(* CODESYS project PLC.project

Project tree, tasks and I/O mapping:
  A_SIM : CODESYS Control Win V3, 3S - Smart Software Solutions GmbH, order no. 305021, version 3.5.10.70
    application PE
      libraries: Standard, * (System); MemoryUtils, * (3S - Smart Software Solutions GmbH); SysTime, 3.5.9.0 (System); PE Core, 0.0.0.23 (ProdexSys); PE User, 0.0.0.15 (ProdexSys)
      task DB (cyclic, interval t#10ms, priority 1) calls DB
      task C100MS (cyclic, interval t#100ms, priority 2) calls C100MS
      task FreeWheel (freewheeling, priority 31) calls SYS, MAIN
      Symbols
      global variables GC
      global variables GVL
      program C100MS [ST]
      program DB [ST]
      program MAIN [ST]: hcb, states, hrb
      program SYS [ST]: updatePointers, initTypes, updateHW, exReadTagsCall, exWriteTagsCall, templateMonitor
      GlobalTypes/
        data type HW
        data type Instances
        data type M
        data type TemplateInstances
        data type TemplateInstancesM
        data type Instructions
        EX/
          data type Exchange
          States/
            data type ValveRegStates
            data type GasFlowRegStates
            data type DriveStates
            data type DriveRegStates
            data type DigOutStates
            data type SensorDigStates
            data type SensorAnStates
            data type PidCStates
            data type HysteresisStates
            data type CascadeStates
            data type HysteresisExStates
            data type WindowExchange
            data type ValveStates
          HCB/
            data type HmiCmd
            data type HmiCmdBuffer
            data type ControlLoop
          HRB/
            data type HmiReadReq
            data type HmiReadRes
            data type HmiReadBuffer
        data type Descriptions
        data type TagsExM
  RLDA : RLDA ARM WinCE (NIL AP), RLDA, ltd., order no. 001, version 3.5.15.10
    application PE
      libraries: Standard, * (System); MemoryUtils, * (3S - Smart Software Solutions GmbH); SysTime, 3.5.9.0 (System); PE Core, 0.0.0.23 (ProdexSys); PE User, 0.0.0.15 (ProdexSys)
      task DB (cyclic, interval t#10ms, priority 1) calls DB
      task FreeWheel (freewheeling, priority 31) calls SYS, MAIN
      task C100MS (cyclic, interval t#100ms, priority 2) calls C100MS
      global variables GC
      global variables GVL
      program C100MS [ST]
      program DB [ST]
      program MAIN [ST]: hcb, states, hrb
      GlobalTypes/
        data type HW
        data type Instances
        data type M
        data type TemplateInstances
        data type TemplateInstancesM
        data type Instructions
        data type Descriptions
        data type TagsExM
        EX/
          data type Exchange
          HCB/
            data type HmiCmd
            data type HmiCmdBuffer
            data type ControlLoop
          HRB/
            data type HmiReadReq
            data type HmiReadRes
            data type HmiReadBuffer
          States/
            data type DriveStates
            data type DriveRegStates
            data type DigOutStates
            data type SensorDigStates
            data type SensorAnStates
            data type PidCStates
            data type HysteresisStates
            data type CascadeStates
            data type HysteresisExStates
            data type WindowExchange
            data type ValveStates
            data type ValveRegStates
            data type GasFlowRegStates
      program SYS [ST]: updateHW, updatePointers, exReadTagsCall, exWriteTagsCall, templateMonitor, initTypes
      Symbols
    Modbus_COM : Modbus COM, 3S - Smart Software Solutions GmbH, version 3.4.0.0
        settings: DataBits = 8; StopBits = 1; ComPort = 2
      Modbus_Master_COM_Port : Modbus Master, COM Port, 3S - Smart Software Solutions GmbH, version 3.5.10.30
        NL_S_16DI : NL(S)-16DI, RLDA, ltd., version 3.5.11.0
            settings: SlaveAddress = 11; ResponseTimeout = 500; UseExtendedFunctionCodes = TRUE
            unmapped channels: Channel 0
        NL_S_8AI_16ch : NL(S)-8AI_16ch, RLDA, ltd., version 3.5.11.0
            settings: SlaveAddress = 10; ResponseTimeout = 500; UseExtendedFunctionCodes = TRUE
            unmapped channels: Channel 0, Channel 1, Channel 2, Channel 3, Channel 4, Channel 5, Channel 6, Channel 7, Channel 8, Channel 9, Channel 10, Channel 11, Channel 12, Channel 13, Channel 14, Channel 15
*)

// A_SIM/PE/GlobalTypes/EX/States/ValveRegStates
TYPE ValveRegStates :
STRUCT
	status : ARRAY[0..GC.VALVE_REG_MAX_IDX]OF DWORD;
	sp : ARRAY[0..GC.VALVE_REG_MAX_IDX]OF REAL;
END_STRUCT
END_TYPE

// A_SIM/PE/GlobalTypes/EX/States/GasFlowRegStates
TYPE GasFlowRegStates :
STRUCT
	status : ARRAY[0..GC.GAS_FLOW_REG_MAX_IDX]OF DWORD;
	sp : ARRAY[0..GC.GAS_FLOW_REG_MAX_IDX]OF REAL;
	pv : ARRAY[0..GC.GAS_FLOW_REG_MAX_IDX]OF REAL;
END_STRUCT
END_TYPE

// A_SIM/PE/GlobalTypes/EX/States/DriveStates
TYPE DriveStates :
STRUCT
	status : ARRAY[0..GC.DRIVE_MAX_IDX]OF DWORD;
END_STRUCT
END_TYPE

// A_SIM/PE/GlobalTypes/EX/States/DriveRegStates
TYPE DriveRegStates :
STRUCT
	status : ARRAY[0..GC.DRIVE_REG_MAX_IDX]OF DWORD;
	sp : ARRAY[0..GC.DRIVE_REG_MAX_IDX]OF REAL;
	pv : ARRAY[0..GC.DRIVE_REG_MAX_IDX]OF REAL;
END_STRUCT
END_TYPE

// A_SIM/PE/GlobalTypes/EX/States/DigOutStates
TYPE DigOutStates :
STRUCT
	status : ARRAY[0..GC.DIG_OUT_MAX_IDX]OF DWORD;
END_STRUCT
END_TYPE

// A_SIM/PE/GlobalTypes/EX/States/SensorDigStates
TYPE SensorDigStates :
STRUCT
	status : ARRAY[0..GC.SENSOR_DIG_MAX_IDX]OF DWORD;
END_STRUCT
END_TYPE

// A_SIM/PE/GlobalTypes/EX/States/SensorAnStates
TYPE SensorAnStates :
STRUCT
	status : ARRAY[0..GC.SENSOR_AN_MAX_IDX]OF DWORD;
	sp : ARRAY[0..GC.SENSOR_AN_MAX_IDX]OF REAL;
	pv : ARRAY[0..GC.SENSOR_AN_MAX_IDX]OF REAL;
END_STRUCT
END_TYPE

// A_SIM/PE/GlobalTypes/EX/States/PidCStates
TYPE PidCStates :
STRUCT
	status : ARRAY[0..GC.PID_C_MAX_IDX]OF DWORD;
	out : ARRAY[0..GC.PID_C_MAX_IDX]OF REAL;
END_STRUCT
END_TYPE

// A_SIM/PE/GlobalTypes/EX/States/HysteresisStates
TYPE HysteresisStates :
STRUCT
	status : ARRAY[0..GC.HYSTERESIS_MAX_IDX]OF DWORD;
	out1 : ARRAY[0..GC.HYSTERESIS_MAX_IDX]OF BOOL;
	out2 : ARRAY[0..GC.HYSTERESIS_MAX_IDX]OF BOOL;
END_STRUCT
END_TYPE

// A_SIM/PE/GlobalTypes/EX/States/CascadeStates
TYPE CascadeStates :
STRUCT
	status : ARRAY[0..GC.REF_MAX_IDX]OF DWORD;
END_STRUCT
END_TYPE

// A_SIM/PE/GlobalTypes/EX/States/HysteresisExStates
TYPE HysteresisExStates :
STRUCT
	status : ARRAY[0..GC.HYSTERESISEX_MAX_IDX]OF DWORD;
	outActuator : ARRAY[0..GC.HYSTERESISEX_MAX_IDX,0..4]OF BOOL;
	out : ARRAY[0..GC.HYSTERESISEX_MAX_IDX]OF BOOL;
END_STRUCT
END_TYPE

// A_SIM/PE/GlobalTypes/EX/States/WindowExchange
TYPE WindowExchange :
STRUCT
	locks : ARRAY[0..GC.WINDOW_MAX_IDX]OF UDINT;
	errors : ARRAY[0..GC.WINDOW_MAX_IDX]OF UDINT;
	status : ARRAY[0..GC.WINDOW_MAX_IDX]OF UDINT;
	workTime : ARRAY[0..GC.WINDOW_MAX_IDX]OF TIME;
END_STRUCT
END_TYPE

// A_SIM/PE/GlobalTypes/HW
TYPE HW :
STRUCT
	di16: ARRAY[0..GC.DI16_MAX_IDX] OF PEU.DI16Instance;
	do16: ARRAY[0..GC.DO16_MAX_IDX] OF PEU.DO16Instance;
	ai16: ARRAY[0..GC.AI16_MAX_IDX] OF PEU.AI16Instance;
	ao4: ARRAY[0..GC.AO4_MAX_IDX] OF PEU.AO4Instance;
END_STRUCT
END_TYPE

// A_SIM/PE/GlobalTypes/Instances
TYPE Instances :
STRUCT
	template: ARRAY[0..PEC.GC.TEMPLATE_MAX_IDX]OF TemplateInstances;
	window : ARRAY[0..PEC.GC.WINDOW_MAX_IDX] OF PEC.WindowInstance;
	parameters : ARRAY[0..PEC.GC.PARAMETERS_MAX_IDX] OF PEC.ParametersInstance;	
	
	valve: ARRAY[0..GC.VALVE_MAX_IDX] OF PEU.ValveInstance;
	valveReg: ARRAY[0..GC.VALVE_REG_MAX_IDX] OF PEU.ValveRegInstance;
	drive: ARRAY[0..GC.DRIVE_MAX_IDX] OF PEU.DriveInstance;
	driveReg: ARRAY[0..GC.DRIVE_REG_MAX_IDX] OF PEU.DriveRegInstance;
	sensorDig : ARRAY[0..GC.SENSOR_DIG_MAX_IDX]OF SensorDigInstance;
	sensorAn : ARRAY[0..GC.SENSOR_AN_MAX_IDX]OF SensorAnInstance;
	pidC : ARRAY[0..GC.PID_C_MAX_IDX]OF PidCInstance;
	hysteresis : ARRAY[0..GC.HYSTERESIS_MAX_IDX]OF HysteresisInstance;
	gasFlowReg : ARRAY[0..GC.GAS_FLOW_REG_MAX_IDX]OF GasFlowRegInstance;
	cascade : ARRAY[0..GC.REF_MAX_IDX]OF CascadeInstance;
	dose : ARRAY[0..GC.DOSE_MAX_IDX]OF DoseInstance;
	profile : ARRAY[0..GC.PROFILE_MAX_IDX]OF ProfileInstance;
	ramp : ARRAY[0..GC.RAMP_MAX_IDX]OF RampInstance;
	route : ARRAY[0..GC.ROUTE_MAX_IDX]OF RouteInstance;
	flip : ARRAY[0..GC.FLIP_MAX_IDX]OF FlipInstance;
	digOut : ARRAY[0..GC.DIG_OUT_MAX_IDX]OF DigOutInstance;
	hysteresisEx : ARRAY[0..GC.HYSTERESISEX_MAX_IDX]OF HysteresisExInstance;
END_STRUCT
END_TYPE

// A_SIM/PE/GlobalTypes/M
TYPE M :
STRUCT
	template : ARRAY[0..PEC.GC.TEMPLATE_MAX_IDX]OF TemplateInstancesM;
	window : ARRAY[0..PEC.GC.WINDOW_MAX_IDX] OF PEC.WindowM;
	parameters : ARRAY[0..PEC.GC.PARAMETERS_MAX_IDX] OF PEC.ParametersM;
	rcpCommon : ARRAY[0..GC.RCP_CALL_INST_MAX_IDX] OF PEC.RcpCommonM;
	rcpStage : ARRAY[0..GC.RCP_CALL_INST_MAX_IDX] OF PEC.RcpStageM;
	rcpStep : ARRAY[0..GC.RCP_CALL_INST_MAX_IDX] OF PEC.RcpStepM;
	di16: ARRAY[0..GC.DI16_MAX_IDX] OF PEU.DI16M;
	do16: ARRAY[0..GC.DO16_MAX_IDX] OF PEU.DO16M;
	ai16: ARRAY[0..GC.AI16_MAX_IDX] OF PEU.AI16M;
	ao4: ARRAY[0..GC.AO4_MAX_IDX] OF PEU.AO4M;
	
	valve: ARRAY[0..GC.VALVE_MAX_IDX] OF PEU.ValveM;
	valveReg: ARRAY[0..GC.VALVE_REG_MAX_IDX] OF PEU.ValveRegM;
	drive: ARRAY[0..GC.DRIVE_MAX_IDX] OF PEU.DriveM;
	driveReg: ARRAY[0..GC.DRIVE_REG_MAX_IDX] OF PEU.DriveRegM;
	sensorDig : ARRAY[0..GC.SENSOR_DIG_MAX_IDX]OF SensorDigM;
	sensorAn : ARRAY[0..GC.SENSOR_AN_MAX_IDX]OF SensorAnM;
	pidC : ARRAY[0..GC.PID_C_MAX_IDX]OF PidCM;
	hysteresis : ARRAY[0..GC.HYSTERESIS_MAX_IDX]OF HysteresisM;
	gasFlowReg : ARRAY[0..GC.GAS_FLOW_REG_MAX_IDX]OF GasFlowRegM;
	cascade : ARRAY[0..GC.REF_MAX_IDX]OF CascadeM;
	dose : ARRAY[0..GC.DOSE_MAX_IDX]OF DoseM;
	profile : ARRAY[0..GC.PROFILE_MAX_IDX]OF ProfileM;
	ramp : ARRAY[0..GC.RAMP_MAX_IDX]OF RampM;
	route : ARRAY[0..GC.ROUTE_MAX_IDX]OF RouteM;
	flip : ARRAY[0..GC.FLIP_MAX_IDX]OF FlipM;
	digOut : ARRAY[0..GC.DIG_OUT_MAX_IDX]OF DigOutM;
	hysteresisEx : ARRAY[0..GC.HYSTERESISEX_MAX_IDX]OF HysteresisExM;
	area: ARRAY[0..GC.AREA_MAX_IDX] OF AreaM;
	
END_STRUCT
END_TYPE

// A_SIM/PE/GlobalTypes/TemplateInstances
TYPE TemplateInstances :
STRUCT
	instance : ARRAY[0..PEC.GC.TEMPLATE_INST_MAX_IDX] OF PEC.TemplateInstance;
END_STRUCT
END_TYPE

// A_SIM/PE/GlobalTypes/TemplateInstancesM
TYPE TemplateInstancesM :
STRUCT
	instance : ARRAY[0..PEC.GC.TEMPLATE_INST_MAX_IDX] OF TemplateInstM;
END_STRUCT
END_TYPE

// A_SIM/PE/GlobalTypes/Instructions
TYPE Instructions :
STRUCT
	edge : ARRAY[0..GC.IEDGE_M_MAX_IDX]OF PEC.IEdgeInstance;
	trig : ARRAY[0..GC.ITRIG_M_MAX_IDX]OF PEC.ITrigInstance;
	timer : ARRAY[0..GC.ITIMER_MAX_IDX]OF PEC.ITimerInstance;
	counter : ARRAY[0..GC.ICOUNTER_MAX_IDX]OF PEC.ICounterInstance;
	pulse : ARRAY[0..GC.IPULSE_MAX_IDX]OF PEC.IPulseInstance;
	rcpCommon : ARRAY[0..GC.RCP_CALL_INST_MAX_IDX] OF PEC.RcpCommonInstance;
	rcpStage : ARRAY[0..GC.RCP_CALL_INST_MAX_IDX] OF PEC.RcpStageInstance;
	rcpStep : ARRAY[0..GC.RCP_CALL_INST_MAX_IDX] OF PEC.RcpStepInstance;
END_STRUCT
END_TYPE

// A_SIM/PE/GlobalTypes/EX/States/ValveStates
TYPE ValveStates :
STRUCT
	status: ARRAY[0..GC.VALVE_MAX_IDX] OF DWORD;
END_STRUCT
END_TYPE

// A_SIM/PE/GlobalTypes/EX/Exchange
TYPE Exchange :
STRUCT	
	hcb: ARRAY[0..GC.HCB_MAX_IDX] OF HmiCmdBuffer;
	hrb: ARRAY[0..GC.HRB_MAX_IDX] OF HmiReadBuffer;
	window : WindowExchange;
	valve : ValveStates;
	valveReg : ValveRegStates;
	gasFlowReg : GasFlowRegStates;
	drive : DriveStates;
	driveReg : DriveRegStates;
	sensorDig : SensorDigStates;
	sensorAn : SensorAnStates;
	pidC : PidCStates;
	hysteresis : HysteresisStates;
	cascade : CascadeStates;
	digOut : DigOutStates;
	hysteresisEx : HysteresisExStates;
END_STRUCT
END_TYPE

// RLDA/PE/GlobalTypes/EX/States/DriveStates
TYPE DriveStates :
STRUCT
	status : ARRAY[0..GC.DRIVE_MAX_IDX]OF DWORD;
END_STRUCT
END_TYPE

// RLDA/PE/GlobalTypes/EX/States/DriveRegStates
TYPE DriveRegStates :
STRUCT
	status : ARRAY[0..GC.DRIVE_REG_MAX_IDX]OF DWORD;
	sp : ARRAY[0..GC.DRIVE_REG_MAX_IDX]OF REAL;
	pv : ARRAY[0..GC.DRIVE_REG_MAX_IDX]OF REAL;
END_STRUCT
END_TYPE

// RLDA/PE/GlobalTypes/EX/States/DigOutStates
TYPE DigOutStates :
STRUCT
	status : ARRAY[0..GC.DIG_OUT_MAX_IDX]OF DWORD;
END_STRUCT
END_TYPE

// RLDA/PE/GlobalTypes/EX/States/SensorDigStates
TYPE SensorDigStates :
STRUCT
	status : ARRAY[0..GC.SENSOR_DIG_MAX_IDX]OF DWORD;
END_STRUCT
END_TYPE

// RLDA/PE/GlobalTypes/EX/States/SensorAnStates
TYPE SensorAnStates :
STRUCT
	status : ARRAY[0..GC.SENSOR_AN_MAX_IDX]OF DWORD;
	sp : ARRAY[0..GC.SENSOR_AN_MAX_IDX]OF REAL;
	pv : ARRAY[0..GC.SENSOR_AN_MAX_IDX]OF REAL;
END_STRUCT
END_TYPE

// RLDA/PE/GlobalTypes/EX/States/PidCStates
TYPE PidCStates :
STRUCT
	status : ARRAY[0..GC.PID_C_MAX_IDX]OF DWORD;
	out : ARRAY[0..GC.PID_C_MAX_IDX]OF REAL;
END_STRUCT
END_TYPE

// RLDA/PE/GlobalTypes/EX/States/HysteresisStates
TYPE HysteresisStates :
STRUCT
	status : ARRAY[0..GC.HYSTERESIS_MAX_IDX]OF DWORD;
	out1 : ARRAY[0..GC.HYSTERESIS_MAX_IDX]OF BOOL;
	out2 : ARRAY[0..GC.HYSTERESIS_MAX_IDX]OF BOOL;
END_STRUCT
END_TYPE

// RLDA/PE/GlobalTypes/EX/States/CascadeStates
TYPE CascadeStates :
STRUCT
	status : ARRAY[0..GC.REF_MAX_IDX]OF DWORD;
END_STRUCT
END_TYPE

// RLDA/PE/GlobalTypes/EX/States/HysteresisExStates
TYPE HysteresisExStates :
STRUCT
	status : ARRAY[0..GC.HYSTERESISEX_MAX_IDX]OF DWORD;
	outActuator : ARRAY[0..GC.HYSTERESISEX_MAX_IDX,0..4]OF BOOL;
	out : ARRAY[0..GC.HYSTERESISEX_MAX_IDX]OF BOOL;
END_STRUCT
END_TYPE

// RLDA/PE/GlobalTypes/EX/States/WindowExchange
TYPE WindowExchange :
STRUCT
	locks : ARRAY[0..GC.WINDOW_MAX_IDX]OF UDINT;
	errors : ARRAY[0..GC.WINDOW_MAX_IDX]OF UDINT;
	status : ARRAY[0..GC.WINDOW_MAX_IDX]OF UDINT;
	workTime : ARRAY[0..GC.WINDOW_MAX_IDX]OF TIME;
END_STRUCT
END_TYPE

// RLDA/PE/GlobalTypes/EX/States/ValveStates
TYPE ValveStates :
STRUCT
	status: ARRAY[0..GC.VALVE_MAX_IDX] OF DWORD;
END_STRUCT
END_TYPE

// RLDA/PE/GlobalTypes/EX/Exchange
TYPE Exchange :
STRUCT	
	hcb: ARRAY[0..GC.HCB_MAX_IDX] OF HmiCmdBuffer;
	hrb: ARRAY[0..GC.HRB_MAX_IDX] OF HmiReadBuffer;
	window : WindowExchange;
	valve : ValveStates;
	valveReg : ValveRegStates;
	gasFlowReg : GasFlowRegStates;
	drive : DriveStates;
	driveReg : DriveRegStates;
	sensorDig : SensorDigStates;
	sensorAn : SensorAnStates;
	pidC : PidCStates;
	hysteresis : HysteresisStates;
	cascade : CascadeStates;
	digOut : DigOutStates;
	hysteresisEx : HysteresisExStates;
END_STRUCT
END_TYPE

// RLDA/PE/GlobalTypes/EX/HCB/HmiCmd
TYPE HmiCmd :
STRUCT
	cId: UINT := 0;
	iId: UINT := 0;
	fc: UINT := 0;
	exId: UINT := 0;
	data: DWORD := 0;
END_STRUCT
END_TYPE

// RLDA/PE/GlobalTypes/EX/HCB/HmiCmdBuffer
TYPE HmiCmdBuffer :
STRUCT
	cLoop: ControlLoop;
	count: UINT := 0;
	cmd: ARRAY[0..GC.HC_BUFFER_MAX_IDX] OF HmiCmd;
END_STRUCT
END_TYPE

// RLDA/PE/GlobalTypes/EX/HCB/ControlLoop
TYPE ControlLoop :
STRUCT
	toPlc: UINT := 0;
	fromPlc: UINT := 0;
END_STRUCT
END_TYPE

// RLDA/PE/GlobalTypes/EX/HRB/HmiReadReq
TYPE HmiReadReq :
STRUCT
	cId: UINT := 0;
	iId: UINT := 0;
	fc: UINT := 0;
	exId: UINT := 0;
END_STRUCT
END_TYPE

// RLDA/PE/GlobalTypes/EX/HRB/HmiReadRes
TYPE HmiReadRes :
STRUCT
	val: ARRAY[0..3] OF UDINT;
END_STRUCT
END_TYPE

// RLDA/PE/GlobalTypes/EX/HRB/HmiReadBuffer
TYPE HmiReadBuffer :
STRUCT
	cLoop: ControlLoop;
	count: UINT := 0;
	req: ARRAY[0..GC.HR_BUFFER_MAX_IDX] OF HmiReadReq;
	res: ARRAY[0..GC.HR_BUFFER_MAX_IDX] OF HmiReadRes;
END_STRUCT
END_TYPE

// RLDA/PE/GlobalTypes/HW
TYPE HW :
STRUCT
	di16: ARRAY[0..GC.DI16_MAX_IDX] OF PEU.DI16Instance;
	do16: ARRAY[0..GC.DO16_MAX_IDX] OF PEU.DO16Instance;
	ai16: ARRAY[0..GC.AI16_MAX_IDX] OF PEU.AI16Instance;
	ao4: ARRAY[0..GC.AO4_MAX_IDX] OF PEU.AO4Instance;
END_STRUCT
END_TYPE

// RLDA/PE/GlobalTypes/Instances
TYPE Instances :
STRUCT
	template: ARRAY[0..PEC.GC.TEMPLATE_MAX_IDX]OF TemplateInstances;
	window : ARRAY[0..PEC.GC.WINDOW_MAX_IDX] OF PEC.WindowInstance;
	parameters : ARRAY[0..PEC.GC.PARAMETERS_MAX_IDX] OF PEC.ParametersInstance;	
	
	valve: ARRAY[0..GC.VALVE_MAX_IDX] OF PEU.ValveInstance;
	valveReg: ARRAY[0..GC.VALVE_REG_MAX_IDX] OF PEU.ValveRegInstance;
	drive: ARRAY[0..GC.DRIVE_MAX_IDX] OF PEU.DriveInstance;
	driveReg: ARRAY[0..GC.DRIVE_REG_MAX_IDX] OF PEU.DriveRegInstance;
	sensorDig : ARRAY[0..GC.SENSOR_DIG_MAX_IDX]OF SensorDigInstance;
	sensorAn : ARRAY[0..GC.SENSOR_AN_MAX_IDX]OF SensorAnInstance;
	pidC : ARRAY[0..GC.PID_C_MAX_IDX]OF PidCInstance;
	hysteresis : ARRAY[0..GC.HYSTERESIS_MAX_IDX]OF HysteresisInstance;
	gasFlowReg : ARRAY[0..GC.GAS_FLOW_REG_MAX_IDX]OF GasFlowRegInstance;
	cascade : ARRAY[0..GC.REF_MAX_IDX]OF CascadeInstance;
	dose : ARRAY[0..GC.DOSE_MAX_IDX]OF DoseInstance;
	profile : ARRAY[0..GC.PROFILE_MAX_IDX]OF ProfileInstance;
	ramp : ARRAY[0..GC.RAMP_MAX_IDX]OF RampInstance;
	route : ARRAY[0..GC.ROUTE_MAX_IDX]OF RouteInstance;
	flip : ARRAY[0..GC.FLIP_MAX_IDX]OF FlipInstance;
	digOut : ARRAY[0..GC.DIG_OUT_MAX_IDX]OF DigOutInstance;
	hysteresisEx : ARRAY[0..GC.HYSTERESISEX_MAX_IDX]OF HysteresisExInstance;
END_STRUCT
END_TYPE

// RLDA/PE/GlobalTypes/M
TYPE M :
STRUCT
	template : ARRAY[0..PEC.GC.TEMPLATE_MAX_IDX]OF TemplateInstancesM;
	window : ARRAY[0..PEC.GC.WINDOW_MAX_IDX] OF PEC.WindowM;
	parameters : ARRAY[0..PEC.GC.PARAMETERS_MAX_IDX] OF PEC.ParametersM;
	rcpCommon : ARRAY[0..GC.RCP_CALL_INST_MAX_IDX] OF PEC.RcpCommonM;
	rcpStage : ARRAY[0..GC.RCP_CALL_INST_MAX_IDX] OF PEC.RcpStageM;
	rcpStep : ARRAY[0..GC.RCP_CALL_INST_MAX_IDX] OF PEC.RcpStepM;
	di16: ARRAY[0..GC.DI16_MAX_IDX] OF PEU.DI16M;
	do16: ARRAY[0..GC.DO16_MAX_IDX] OF PEU.DO16M;
	ai16: ARRAY[0..GC.AI16_MAX_IDX] OF PEU.AI16M;
	ao4: ARRAY[0..GC.AO4_MAX_IDX] OF PEU.AO4M;
	
	valve: ARRAY[0..GC.VALVE_MAX_IDX] OF PEU.ValveM;
	valveReg: ARRAY[0..GC.VALVE_REG_MAX_IDX] OF PEU.ValveRegM;
	drive: ARRAY[0..GC.DRIVE_MAX_IDX] OF PEU.DriveM;
	driveReg: ARRAY[0..GC.DRIVE_REG_MAX_IDX] OF PEU.DriveRegM;
	sensorDig : ARRAY[0..GC.SENSOR_DIG_MAX_IDX]OF SensorDigM;
	sensorAn : ARRAY[0..GC.SENSOR_AN_MAX_IDX]OF SensorAnM;
	pidC : ARRAY[0..GC.PID_C_MAX_IDX]OF PidCM;
	hysteresis : ARRAY[0..GC.HYSTERESIS_MAX_IDX]OF HysteresisM;
	gasFlowReg : ARRAY[0..GC.GAS_FLOW_REG_MAX_IDX]OF GasFlowRegM;
	cascade : ARRAY[0..GC.REF_MAX_IDX]OF CascadeM;
	dose : ARRAY[0..GC.DOSE_MAX_IDX]OF DoseM;
	profile : ARRAY[0..GC.PROFILE_MAX_IDX]OF ProfileM;
	ramp : ARRAY[0..GC.RAMP_MAX_IDX]OF RampM;
	route : ARRAY[0..GC.ROUTE_MAX_IDX]OF RouteM;
	flip : ARRAY[0..GC.FLIP_MAX_IDX]OF FlipM;
	digOut : ARRAY[0..GC.DIG_OUT_MAX_IDX]OF DigOutM;
	hysteresisEx : ARRAY[0..GC.HYSTERESISEX_MAX_IDX]OF HysteresisExM;
	area: ARRAY[0..GC.AREA_MAX_IDX] OF AreaM;
	
END_STRUCT
END_TYPE

// RLDA/PE/GlobalTypes/TemplateInstances
TYPE TemplateInstances :
STRUCT
	instance : ARRAY[0..PEC.GC.TEMPLATE_INST_MAX_IDX] OF PEC.TemplateInstance;
END_STRUCT
END_TYPE

// RLDA/PE/GlobalTypes/TemplateInstancesM
TYPE TemplateInstancesM :
STRUCT
	instance : ARRAY[0..PEC.GC.TEMPLATE_INST_MAX_IDX] OF TemplateInstM;
END_STRUCT
END_TYPE

// RLDA/PE/GlobalTypes/Instructions
TYPE Instructions :
STRUCT
	edge : ARRAY[0..GC.IEDGE_M_MAX_IDX]OF PEC.IEdgeInstance;
	trig : ARRAY[0..GC.ITRIG_M_MAX_IDX]OF PEC.ITrigInstance;
	timer : ARRAY[0..GC.ITIMER_MAX_IDX]OF PEC.ITimerInstance;
	counter : ARRAY[0..GC.ICOUNTER_MAX_IDX]OF PEC.ICounterInstance;
	pulse : ARRAY[0..GC.IPULSE_MAX_IDX]OF PEC.IPulseInstance;
	rcpCommon : ARRAY[0..GC.RCP_CALL_INST_MAX_IDX] OF PEC.RcpCommonInstance;
	rcpStage : ARRAY[0..GC.RCP_CALL_INST_MAX_IDX] OF PEC.RcpStageInstance;
	rcpStep : ARRAY[0..GC.RCP_CALL_INST_MAX_IDX] OF PEC.RcpStepInstance;
END_STRUCT
END_TYPE

// RLDA/PE/GlobalTypes/Descriptions
TYPE Descriptions :
STRUCT
	template: TemplateInstance;
	window : WindowInstance;
	parameters : ParametersInstance;
	valve: ValveInstance;
	valveReg: ValveRegInstance;
	drive: DriveInstance;
	driveReg: DriveRegInstance;
	sensorDig : SensorDigInstance;
	sensorAn : SensorAnInstance;
	pidC : PidCInstance;
	hysteresis : HysteresisInstance;
	gasFlowReg : GasFlowRegInstance;
	cascade : CascadeInstance;
	dose : DoseInstance;
	profile : ProfileInstance;
	ramp : RampInstance;
	route : RouteInstance;
	flip : FlipInstance;
	digOut : DigOutInstance;
	hysteresisEx : HysteresisExInstance;
	timer : ITimerInstance;
	counter : ICounterInstance;
	edge : IEdgeInstance;
	pulse : IPulseInstance;
	trig : ITrigInstance;
	
	di16: PEU.DI16Instance;
	do16: PEU.DO16Instance;
	ai16: PEU.AI16Instance;
	ao4: PEU.AO4Instance;
END_STRUCT
END_TYPE

// RLDA/PE/GlobalTypes/TagsExM
TYPE TagsExM :
STRUCT
	readState: USINT;
	readResetTimeout: TON;
	writeState: USINT;
	writeResetTimeout: TON; 
END_STRUCT
END_TYPE

// RLDA/PE/GlobalTypes/EX/States/ValveRegStates
TYPE ValveRegStates :
STRUCT
	status : ARRAY[0..GC.VALVE_REG_MAX_IDX]OF DWORD;
	sp : ARRAY[0..GC.VALVE_REG_MAX_IDX]OF REAL;
END_STRUCT
END_TYPE

// RLDA/PE/GlobalTypes/EX/States/GasFlowRegStates
TYPE GasFlowRegStates :
STRUCT
	status : ARRAY[0..GC.GAS_FLOW_REG_MAX_IDX]OF DWORD;
	sp : ARRAY[0..GC.GAS_FLOW_REG_MAX_IDX]OF REAL;
	pv : ARRAY[0..GC.GAS_FLOW_REG_MAX_IDX]OF REAL;
END_STRUCT
END_TYPE

// A_SIM/PE/GlobalTypes/Descriptions
TYPE Descriptions :
STRUCT
	template: TemplateInstance;
	window : WindowInstance;
	parameters : ParametersInstance;
	valve: ValveInstance;
	valveReg: ValveRegInstance;
	drive: DriveInstance;
	driveReg: DriveRegInstance;
	sensorDig : SensorDigInstance;
	sensorAn : SensorAnInstance;
	pidC : PidCInstance;
	hysteresis : HysteresisInstance;
	gasFlowReg : GasFlowRegInstance;
	cascade : CascadeInstance;
	dose : DoseInstance;
	profile : ProfileInstance;
	ramp : RampInstance;
	route : RouteInstance;
	flip : FlipInstance;
	digOut : DigOutInstance;
	hysteresisEx : HysteresisExInstance;
	timer : ITimerInstance;
	counter : ICounterInstance;
	edge : IEdgeInstance;
	pulse : IPulseInstance;
	trig : ITrigInstance;
	
	di16: PEU.DI16Instance;
	do16: PEU.DO16Instance;
	ai16: PEU.AI16Instance;
	ao4: PEU.AO4Instance;
END_STRUCT
END_TYPE

// A_SIM/PE/GlobalTypes/TagsExM
TYPE TagsExM :
STRUCT
	readState: USINT;
	readResetTimeout: TON;
	writeState: USINT;
	writeResetTimeout: TON; 
END_STRUCT
END_TYPE

// A_SIM/PE/GlobalTypes/EX/HCB/HmiCmd
TYPE HmiCmd :
STRUCT
	cId: UINT := 0;
	iId: UINT := 0;
	fc: UINT := 0;
	exId: UINT := 0;
	data: DWORD := 0;
END_STRUCT
END_TYPE

// A_SIM/PE/GlobalTypes/EX/HCB/HmiCmdBuffer
TYPE HmiCmdBuffer :
STRUCT
	cLoop: ControlLoop;
	count: UINT := 0;
	cmd: ARRAY[0..GC.HC_BUFFER_MAX_IDX] OF HmiCmd;
END_STRUCT
END_TYPE

// A_SIM/PE/GlobalTypes/EX/HCB/ControlLoop
TYPE ControlLoop :
STRUCT
	toPlc: UINT := 0;
	fromPlc: UINT := 0;
END_STRUCT
END_TYPE

// A_SIM/PE/GlobalTypes/EX/HRB/HmiReadReq
TYPE HmiReadReq :
STRUCT
	cId: UINT := 0;
	iId: UINT := 0;
	fc: UINT := 0;
	exId: UINT := 0;
END_STRUCT
END_TYPE

// A_SIM/PE/GlobalTypes/EX/HRB/HmiReadRes
TYPE HmiReadRes :
STRUCT
	val: ARRAY[0..3] OF UDINT;
END_STRUCT
END_TYPE

// A_SIM/PE/GlobalTypes/EX/HRB/HmiReadBuffer
TYPE HmiReadBuffer :
STRUCT
	cLoop: ControlLoop;
	count: UINT := 0;
	req: ARRAY[0..GC.HR_BUFFER_MAX_IDX] OF HmiReadReq;
	res: ARRAY[0..GC.HR_BUFFER_MAX_IDX] OF HmiReadRes;
END_STRUCT
END_TYPE

// A_SIM/PE/GC
{attribute 'qualified_only'}
VAR_GLOBAL CONSTANT
	HCB_MAX_IDX: USINT := 3;
	HRB_MAX_IDX: USINT := 0;
	HC_BUFFER_MAX_IDX: UINT := 9;
	HR_BUFFER_MAX_IDX: UINT := 511;
	CW_MAX_IDX: USINT := 7;
	WINDOW_MAX_IDX : UINT := 63;
	IEDGE_M_MAX_IDX : UINT := 1023;
	ITRIG_M_MAX_IDX : UINT := 1023;
	ITIMER_MAX_IDX : UINT := 1023;
	ICOUNTER_MAX_IDX : UINT := 1023;
	IPULSE_MAX_IDX : UINT := 1023;
	VALVE_MAX_IDX : UINT := 149;
	VALVE_REG_MAX_IDX : UINT := 15;
	GAS_FLOW_REG_MAX_IDX : UINT := 15;
	DRIVE_MAX_IDX : UINT := 31;
	DRIVE_REG_MAX_IDX : UINT := 31;
	DIG_OUT_MAX_IDX : UINT := 31;
	PID_C_MAX_IDX : UINT := 127;
	HYSTERESIS_MAX_IDX : UINT := 63;
	REF_MAX_IDX : UINT := 63;
	HYSTERESISEX_MAX_IDX : UINT := 63;
	SENSOR_DIG_MAX_IDX : UINT := 31;
	SENSOR_AN_MAX_IDX : UINT := 63;
	AREA_MAX_IDX : UINT := 9;
	DOSE_MAX_IDX : UINT := 63;
	FLIP_MAX_IDX : UINT := 63;
	ROUTE_MAX_IDX : UINT := 255;
	PROFILE_MAX_IDX : UINT := 63;
	RAMP_MAX_IDX : UINT := 63;
	RCP_CALL_INST_MAX_IDX : USINT := 127;
	
	AI16_MAX_IDX : UINT := 15;
	AO4_MAX_IDX : UINT := 15;
	DI16_MAX_IDX : UINT := 15;
	DO16_MAX_IDX : UINT := 15;
END_VAR

// A_SIM/PE/GVL
{attribute 'qualified_only'}
VAR_GLOBAL
	systemData: PEC.SystemData;
	area: ARRAY[0..GC.AREA_MAX_IDX] OF AreaInstance;
	templates : ARRAY[0..PEC.GC.TEMPLATE_MAX_IDX] OF TemplateBody;
	interfaces : ARRAY[0..PEC.GC.CLASS_MAX_IDX] OF ClassInterface;	
	hw: HW;
	instances: Instances;	
	instructions: Instructions;	
	m: M;
	ex: Exchange;
END_VAR

// RLDA/PE/GC
{attribute 'qualified_only'}
VAR_GLOBAL CONSTANT
	HCB_MAX_IDX: USINT := 3;
	HRB_MAX_IDX: USINT := 0;
	HC_BUFFER_MAX_IDX: UINT := 9;
	HR_BUFFER_MAX_IDX: UINT := 511;
	CW_MAX_IDX: USINT := 7;
	WINDOW_MAX_IDX : UINT := 63;
	IEDGE_M_MAX_IDX : UINT := 1023;
	ITRIG_M_MAX_IDX : UINT := 1023;
	ITIMER_MAX_IDX : UINT := 1023;
	ICOUNTER_MAX_IDX : UINT := 1023;
	IPULSE_MAX_IDX : UINT := 1023;
	VALVE_MAX_IDX : UINT := 149;
	VALVE_REG_MAX_IDX : UINT := 15;
	GAS_FLOW_REG_MAX_IDX : UINT := 15;
	DRIVE_MAX_IDX : UINT := 31;
	DRIVE_REG_MAX_IDX : UINT := 31;
	DIG_OUT_MAX_IDX : UINT := 31;
	PID_C_MAX_IDX : UINT := 127;
	HYSTERESIS_MAX_IDX : UINT := 63;
	REF_MAX_IDX : UINT := 63;
	HYSTERESISEX_MAX_IDX : UINT := 63;
	SENSOR_DIG_MAX_IDX : UINT := 31;
	SENSOR_AN_MAX_IDX : UINT := 63;
	AREA_MAX_IDX : UINT := 9;
	DOSE_MAX_IDX : UINT := 63;
	FLIP_MAX_IDX : UINT := 63;
	ROUTE_MAX_IDX : UINT := 255;
	PROFILE_MAX_IDX : UINT := 63;
	RAMP_MAX_IDX : UINT := 63;
	RCP_CALL_INST_MAX_IDX : USINT := 127;
	
	AI16_MAX_IDX : UINT := 15;
	AO4_MAX_IDX : UINT := 15;
	DI16_MAX_IDX : UINT := 15;
	DO16_MAX_IDX : UINT := 15;
END_VAR

// RLDA/PE/GVL
{attribute 'qualified_only'}
VAR_GLOBAL
	systemData: PEC.SystemData;
	area: ARRAY[0..GC.AREA_MAX_IDX] OF AreaInstance;
	templates : ARRAY[0..PEC.GC.TEMPLATE_MAX_IDX] OF TemplateBody;
	interfaces : ARRAY[0..PEC.GC.CLASS_MAX_IDX] OF ClassInterface;	
	hw: HW;
	instances: Instances;	
	instructions: Instructions;	
	m: M;
	ex: Exchange;
END_VAR

// A_SIM/PE/DB
PROGRAM DB
VAR
	databaseEx: PEC.DatabaseEx;
	database: PEC.Database;
END_VAR

database.pSD := ADR(GVL.systemData);
database.pEx := ADR(databaseEx);
database.pRoot := ADR('..\PJ_DBC\');		
database();

END_PROGRAM

// RLDA/PE/DB
PROGRAM DB
VAR
	databaseEx: PEC.DatabaseEx;
	database: PEC.Database;
END_VAR

database.pSD := ADR(GVL.systemData);
database.pEx := ADR(databaseEx);
database.pRoot := ADR('..\PJ_DBC\');		
database();

END_PROGRAM

// A_SIM/PE/C100MS
PROGRAM C100MS
VAR
	flagsHolder: CallFlags;
	linkHolder: InstanceLink;
	callCounter: UINT := 0;
	c500ms: UINT := 0;
	c1s: UINT := 0;
	c10s: UINT := 0;
	c1m: UINT := 0;
END_VAR

IF(GVL.systemData.rt.control.run)THEN	
	GVL.systemData.rt.state.cyclicOff := FALSE;
	flagsHolder := GVL.systemData.callFlags;
	linkHolder := GVL.systemData.execLink;
	MEMUtils.MemSet(ADR(GVL.systemData.callFlags), 0, SIZEOF(CallFlags));
	GVL.systemData.callFlags.c100ms := TRUE;
	GVL.systemData.callFlags.c500ms := PEC.callPulse(5, c500ms);
	GVL.systemData.callFlags.c1s := PEC.callPulse(10, c1s);
	GVL.systemData.callFlags.c10s := PEC.callPulse(100, c10s);
	GVL.systemData.callFlags.c1m := PEC.callPulse(600, c1m);
	
	PEC.exec(ADR(GVL.systemData));
	
	GVL.systemData.execLink := linkHolder;
	GVL.systemData.callFlags := flagsHolder;
	callCounter := callCounter + 1;
ELSE 
	GVL.systemData.rt.state.cyclicOff := TRUE;	
END_IF;

END_PROGRAM

// RLDA/PE/C100MS
PROGRAM C100MS
VAR
	flagsHolder: CallFlags;
	linkHolder: InstanceLink;
	callCounter: UINT := 0;
	c500ms: UINT := 0;
	c1s: UINT := 0;
	c10s: UINT := 0;
	c1m: UINT := 0;
END_VAR

IF(GVL.systemData.rt.control.run)THEN	
	GVL.systemData.rt.state.cyclicOff := FALSE;
	flagsHolder := GVL.systemData.callFlags;
	linkHolder := GVL.systemData.execLink;
	MEMUtils.MemSet(ADR(GVL.systemData.callFlags), 0, SIZEOF(CallFlags));
	GVL.systemData.callFlags.c100ms := TRUE;
	GVL.systemData.callFlags.c500ms := PEC.callPulse(5, c500ms);
	GVL.systemData.callFlags.c1s := PEC.callPulse(10, c1s);
	GVL.systemData.callFlags.c10s := PEC.callPulse(100, c10s);
	GVL.systemData.callFlags.c1m := PEC.callPulse(600, c1m);
	
	PEC.exec(ADR(GVL.systemData));
	
	GVL.systemData.execLink := linkHolder;
	GVL.systemData.callFlags := flagsHolder;
	callCounter := callCounter + 1;
ELSE 
	GVL.systemData.rt.state.cyclicOff := TRUE;	
END_IF;

END_PROGRAM

// A_SIM/PE/SYS
PROGRAM SYS
VAR	
	registry: PEC.Registry;
	templateMonitorEx : TemplateMonitorEx;
	id: UINT;
	descriptions: Descriptions;
	readTagsEx: PEC.ReadTagsEx;
	writeTagsEx: PEC.WriteTagsEx;	
	xInit: BOOL := TRUE;
	xReq: BOOL := FALSE;
	tagsExM: TagsExM;
	persistList: PersistList;
END_VAR

GVL.systemData.xFalse := FALSE;
GVL.systemData.xTrue := TRUE;
GVL.systemData.db.control.enable := TRUE;
GVL.systemData.rt.control.run := GVL.systemData.db.state.run;

initTypes();
updatePointers();
exReadTagsCall();
exWriteTagsCall();
templateMonitor();

(*IF GVL.systemData.db.state.run THEN 
	updateHW();	
	
	id := 158;
	registry.instances[id - 1].count := 1;
	registry.instances[id - 1].name := 'DO16';
	registry.instances[id - 1].flags.main := TRUE;
	registry.instances[id - 1].sum := 629;
	
	id := 159;
	registry.instances[id - 1].count := 1;
	registry.instances[id - 1].name := 'AI16';
	registry.instances[id - 1].flags.main := TRUE;
	registry.instances[id - 1].sum := 659;
	
	id := 200;
	registry.instances[id - 1].count := 5;
	registry.instances[id - 1].name := 'Valve';
	registry.instances[id - 1].flags.main := TRUE;
	registry.instances[id - 1].sum := 7287;	
END_IF*)

METHOD PUBLIC updatePointers
VAR_INPUT
END_VAR
VAR
	id: UINT;
END_VAR
//SYSTEM DATA
GVL.systemData.pStack := 0;
GVL.systemData.pRegistry := ADR(SYS.registry);
GVL.systemData.pRecipes := 0;
GVL.systemData.pTemplates := ADR(GVL.templates);
GVL.systemData.pInterfaces := ADR(GVL.interfaces);
GVL.systemData.pTemplateMonitorEx := ADR(templateMonitorEx);
GVL.systemData.pAcc := 0;
GVL.systemData.pSlaves := 0;
GVL.systemData.pPersistList := ADR(persistList);

FOR id := 1 TO PEC.GC.TEMPLATE_MAX_IDX + 1 DO
		registry.pointers[id - 1].pFC := ADR(Template);
		registry.pointers[id - 1].pB := ADR(GVL.templates[id - 1]);
		registry.pointers[id - 1].vpI._pointer := ADR(GVL.instances.template[id - 1]);
		registry.pointers[id - 1].vpI.size := SIZEOF(TemplateInstance);
		registry.pointers[id - 1].vpM._pointer := ADR(GVL.m.template[id - 1]);
		registry.pointers[id - 1].vpM.size := SIZEOF(TemplateInstM);
END_FOR

//INSTRUCTIONS AND SYSTEM CLASSES
id := 150;	//IEdge
registry.pointers[id - 1].pFC := ADR(PEC.IEdge);
registry.pointers[id - 1].pB := 0;
registry.pointers[id - 1].vpI._pointer := ADR(GVL.instructions.edge);
registry.pointers[id - 1].vpI.size := SIZEOF(PEC.IEdgeInstance);
registry.pointers[id - 1].vpM._pointer := 0;
registry.pointers[id - 1].vpM.size := 0;

id := 151; //ITrig
registry.pointers[id - 1].pFC := ADR(PEC.ITrig);
registry.pointers[id - 1].pB := 0;
registry.pointers[id - 1].vpI._pointer := ADR(GVL.instructions.trig);
registry.pointers[id - 1].vpI.size := SIZEOF(PEC.ITrigInstance);
registry.pointers[id - 1].vpM._pointer := 0;
registry.pointers[id - 1].vpM.size := 0;

id := 152; //ITimer
registry.pointers[id - 1].pFC := ADR(PEC.ITimer);
registry.pointers[id - 1].pB := 0;
registry.pointers[id - 1].vpI._pointer := ADR(GVL.instructions.timer);
registry.pointers[id - 1].vpI.size := SIZEOF(PEC.ITimerInstance);
registry.pointers[id - 1].vpM._pointer := 0;
registry.pointers[id - 1].vpM.size := 0;

id := 153; //ICounter
registry.pointers[id - 1].pFC := ADR(PEC.ICounter);
registry.pointers[id - 1].pB := 0;
registry.pointers[id - 1].vpI._pointer := ADR(GVL.instructions.counter);
registry.pointers[id - 1].vpI.size := SIZEOF(PEC.ICounterInstance);
registry.pointers[id - 1].vpM._pointer := 0;
registry.pointers[id - 1].vpM.size := 0;

id := 155; //DigOut
registry.pointers[id - 1].pFC := ADR(PEU.DigOut);
registry.pointers[id - 1].pB := 0;
registry.pointers[id - 1].vpI._pointer := ADR(GVL.instances.digOut);
registry.pointers[id - 1].vpI.size := SIZEOF(PEU.DigOutInstance);
registry.pointers[id - 1].vpM._pointer := ADR(GVL.m.digOut);;
registry.pointers[id - 1].vpM.size := SIZEOF(PEU.digOutM);

id := 157; //DI16
registry.pointers[id - 1].pFC := ADR(PEU.DI16);
registry.pointers[id - 1].pB := 0;
registry.pointers[id - 1].vpI._pointer := ADR(GVL.hw.di16);
registry.pointers[id - 1].vpI.size := SIZEOF(PEU.DI16Instance);
registry.pointers[id - 1].vpM._pointer := ADR(GVL.m.di16);;
registry.pointers[id - 1].vpM.size := SIZEOF(PEU.DI16M);

id := 158; //DO16
registry.pointers[id - 1].pFC := ADR(PEU.DO16);
registry.pointers[id - 1].pB := 0;
registry.pointers[id - 1].vpI._pointer := ADR(GVL.hw.do16);
registry.pointers[id - 1].vpI.size := SIZEOF(PEU.DO16Instance);
registry.pointers[id - 1].vpM._pointer := ADR(GVL.m.do16);;
registry.pointers[id - 1].vpM.size := SIZEOF(PEU.DO16M);

id := 159; //AI16
registry.pointers[id - 1].pFC := ADR(PEU.AI16);
registry.pointers[id - 1].pB := 0;
registry.pointers[id - 1].vpI._pointer := ADR(GVL.hw.ai16);
registry.pointers[id - 1].vpI.size := SIZEOF(PEU.AI16Instance);
registry.pointers[id - 1].vpM._pointer := ADR(GVL.m.ai16);;
registry.pointers[id - 1].vpM.size := SIZEOF(PEU.AI16M);

id := 160; //AO4
registry.pointers[id - 1].pFC := ADR(PEU.AO4);
registry.pointers[id - 1].pB := 0;
registry.pointers[id - 1].vpI._pointer := ADR(GVL.hw.ao4);
registry.pointers[id - 1].vpI.size := SIZEOF(PEU.AO4Instance);
registry.pointers[id - 1].vpM._pointer := ADR(GVL.m.ao4);;
registry.pointers[id - 1].vpM.size := SIZEOF(PEU.AO4M);


id := 161; //RcpCommon	
registry.pointers[id - 1].pFC := ADR(PEC.RcpCommon);
registry.pointers[id - 1].pB := 0;
registry.pointers[id - 1].vpI._pointer := ADR(GVL.instructions.rcpCommon);
registry.pointers[id - 1].vpI.size := SIZEOF(PEC.RcpCommonInstance);
registry.pointers[id - 1].vpM._pointer := ADR(GVL.m.rcpCommon);
registry.pointers[id - 1].vpM.size := SIZEOF(PEC.RcpCommonM);

id := 162; //RcpStage
registry.pointers[id - 1].pFC := ADR(PEC.RcpStage);
registry.pointers[id - 1].pB := 0;
registry.pointers[id - 1].vpI._pointer := ADR(GVL.instructions.rcpStage);
registry.pointers[id - 1].vpI.size := SIZEOF(PEC.RcpStageInstance);
registry.pointers[id - 1].vpM._pointer := ADR(GVL.m.rcpStage);
registry.pointers[id - 1].vpM.size := SIZEOF(PEC.RcpStageM);

id := 163; //RcpStep
registry.pointers[id - 1].pFC := ADR(PEC.RcpStep);
registry.pointers[id - 1].pB := 0;
registry.pointers[id - 1].vpI._pointer := ADR(GVL.instructions.rcpStep);
registry.pointers[id - 1].vpI.size := SIZEOF(PEC.RcpStepInstance);
registry.pointers[id - 1].vpM._pointer := ADR(GVL.m.rcpStep);
registry.pointers[id - 1].vpM.size := SIZEOF(PEC.RcpStepM);

id := 164; //Window
registry.pointers[id - 1].pFC := ADR(PEC.Window);
registry.pointers[id - 1].pB := 0;
registry.pointers[id - 1].vpI._pointer := ADR(GVL.instances.window);
registry.pointers[id - 1].vpI.size := SIZEOF(PEC.WindowInstance);
registry.pointers[id - 1].vpM._pointer := ADR(GVL.m.window);
registry.pointers[id - 1].vpM.size := SIZEOF(PEC.WindowM);

id := 165; //Parameters
registry.pointers[id - 1].pFC := ADR(PEC.Parameters);
registry.pointers[id - 1].pB := 0;
registry.pointers[id - 1].vpI._pointer := ADR(GVL.instances.parameters);
registry.pointers[id - 1].vpI.size := SIZEOF(PEC.ParametersInstance);
registry.pointers[id - 1].vpM._pointer := ADR(GVL.m.parameters);
registry.pointers[id - 1].vpM.size := SIZEOF(PEC.ParametersM);

id := 166; //IPulse
registry.pointers[id - 1].pFC := ADR(PEC.IPulse);
registry.pointers[id - 1].pB := 0;
registry.pointers[id - 1].vpI._pointer := ADR(GVL.instructions.pulse);
registry.pointers[id - 1].vpI.size := SIZEOF(PEC.IPulseInstance);
registry.pointers[id - 1].vpM._pointer := 0;
registry.pointers[id - 1].vpM.size := 0;

//USER TYPES
id := 200;	
registry.pointers[id - 1].pFC := ADR(PEU.Valve);
registry.pointers[id - 1].pB := 0;
registry.pointers[id - 1].vpI._pointer := ADR(GVL.instances.valve);
registry.pointers[id - 1].vpI.size := SIZEOF(PEU.ValveInstance);
registry.pointers[id - 1].vpM._pointer := ADR(GVL.m.valve);
registry.pointers[id - 1].vpM.size := SIZEOF(PEU.ValveM);

id := 201;	
registry.pointers[id - 1].pFC := ADR(PEU.ValveReg);
registry.pointers[id - 1].pB := 0;
registry.pointers[id - 1].vpI._pointer := ADR(GVL.instances.valveReg);
registry.pointers[id - 1].vpI.size := SIZEOF(PEU.ValveRegInstance);
registry.pointers[id - 1].vpM._pointer := ADR(GVL.m.valveReg);
registry.pointers[id - 1].vpM.size := SIZEOF(PEU.ValveRegM);

id := 202;	
registry.pointers[id - 1].pFC := ADR(PEU.Drive);
registry.pointers[id - 1].pB := 0;
registry.pointers[id - 1].vpI._pointer := ADR(GVL.instances.drive);
registry.pointers[id - 1].vpI.size := SIZEOF(PEU.DriveInstance);
registry.pointers[id - 1].vpM._pointer := ADR(GVL.m.drive);
registry.pointers[id - 1].vpM.size := SIZEOF(PEU.DriveM);

id := 203;	
registry.pointers[id - 1].pFC := ADR(PEU.DriveReg);
registry.pointers[id - 1].pB := 0;
registry.pointers[id - 1].vpI._pointer := ADR(GVL.instances.driveReg);
registry.pointers[id - 1].vpI.size := SIZEOF(PEU.DriveRegInstance);
registry.pointers[id - 1].vpM._pointer := ADR(GVL.m.driveReg);
registry.pointers[id - 1].vpM.size := SIZEOF(PEU.DriveRegM);

id := 204;	
registry.pointers[id - 1].pFC := ADR(PEU.SensorDig);
registry.pointers[id - 1].pB := 0;
registry.pointers[id - 1].vpI._pointer := ADR(GVL.instances.sensorDig);
registry.pointers[id - 1].vpI.size := SIZEOF(PEU.SensorDigInstance);
registry.pointers[id - 1].vpM._pointer := ADR(GVL.m.sensorDig);
registry.pointers[id - 1].vpM.size := SIZEOF(PEU.SensorDigM);

id := 205;	
registry.pointers[id - 1].pFC := ADR(PEU.SensorAn);
registry.pointers[id - 1].pB := 0;
registry.pointers[id - 1].vpI._pointer := ADR(GVL.instances.sensorAn);
registry.pointers[id - 1].vpI.size := SIZEOF(PEU.SensorAnInstance);
registry.pointers[id - 1].vpM._pointer := ADR(GVL.m.sensorAn);
registry.pointers[id - 1].vpM.size := SIZEOF(PEU.SensorAnM);

id := 206;


id := 207;	
registry.pointers[id - 1].pFC := ADR(PEU.Hysteresis);
registry.pointers[id - 1].pB := 0;
registry.pointers[id - 1].vpI._pointer := ADR(GVL.instances.hysteresis);
registry.pointers[id - 1].vpI.size := SIZEOF(PEU.HysteresisInstance);
registry.pointers[id - 1].vpM._pointer := ADR(GVL.m.hysteresis);
registry.pointers[id - 1].vpM.size := SIZEOF(PEU.HysteresisM);

id := 208;	
registry.pointers[id - 1].pFC := ADR(PEU.GasFlowReg);
registry.pointers[id - 1].pB := 0;
registry.pointers[id - 1].vpI._pointer := ADR(GVL.instances.gasFlowReg);
registry.pointers[id - 1].vpI.size := SIZEOF(PEU.GasFlowRegInstance);
registry.pointers[id - 1].vpM._pointer := ADR(GVL.m.gasFlowReg);
registry.pointers[id - 1].vpM.size := SIZEOF(PEU.GasFlowRegM);

id := 209;	
registry.pointers[id - 1].pFC := ADR(PEU.Cascade);
registry.pointers[id - 1].pB := 0;
registry.pointers[id - 1].vpI._pointer := ADR(GVL.instances.cascade);
registry.pointers[id - 1].vpI.size := SIZEOF(PEU.CascadeInstance);
registry.pointers[id - 1].vpM._pointer := ADR(GVL.m.cascade);
registry.pointers[id - 1].vpM.size := SIZEOF(PEU.CascadeM);

id := 210;	
registry.pointers[id - 1].pFC := ADR(PEU.Dose);
registry.pointers[id - 1].pB := 0;
registry.pointers[id - 1].vpI._pointer := ADR(GVL.instances.dose);
registry.pointers[id - 1].vpI.size := SIZEOF(PEU.DoseInstance);
registry.pointers[id - 1].vpM._pointer := ADR(GVL.m.dose);
registry.pointers[id - 1].vpM.size := SIZEOF(PEU.DoseM);

id := 211;	
registry.pointers[id - 1].pFC := ADR(PEU.Profile);
registry.pointers[id - 1].pB := 0;
registry.pointers[id - 1].vpI._pointer := ADR(GVL.instances.profile);
registry.pointers[id - 1].vpI.size := SIZEOF(PEU.ProfileInstance);
registry.pointers[id - 1].vpM._pointer := ADR(GVL.m.profile);
registry.pointers[id - 1].vpM.size := SIZEOF(PEU.ProfileM);

id := 212;	
registry.pointers[id - 1].pFC := ADR(PEU.Ramp);
registry.pointers[id - 1].pB := 0;
registry.pointers[id - 1].vpI._pointer := ADR(GVL.instances.ramp);
registry.pointers[id - 1].vpI.size := SIZEOF(PEU.RampInstance);
registry.pointers[id - 1].vpM._pointer := ADR(GVL.m.ramp);
registry.pointers[id - 1].vpM.size := SIZEOF(PEU.RampM);

id := 213;	
registry.pointers[id - 1].pFC := ADR(PEU.Route);
registry.pointers[id - 1].pB := 0;
registry.pointers[id - 1].vpI._pointer := ADR(GVL.instances.route);
registry.pointers[id - 1].vpI.size := SIZEOF(PEU.RouteInstance);
registry.pointers[id - 1].vpM._pointer := ADR(GVL.m.route);
registry.pointers[id - 1].vpM.size := SIZEOF(PEU.RouteM);

id := 214;	
registry.pointers[id - 1].pFC := ADR(PEU.Flip);
registry.pointers[id - 1].pB := 0;
registry.pointers[id - 1].vpI._pointer := ADR(GVL.instances.flip);
registry.pointers[id - 1].vpI.size := SIZEOF(PEU.FlipInstance);
registry.pointers[id - 1].vpM._pointer := ADR(GVL.m.flip);
registry.pointers[id - 1].vpM.size := SIZEOF(PEU.FlipM);

id := 219;	
registry.pointers[id - 1].pFC := ADR(PEU.Area);
registry.pointers[id - 1].pB := 0;
registry.pointers[id - 1].vpI._pointer := ADR(GVL.area);
registry.pointers[id - 1].vpI.size := SIZEOF(PEU.AreaInstance);
registry.pointers[id - 1].vpM._pointer := ADR(GVL.m.area);
registry.pointers[id - 1].vpM.size := SIZEOF(PEU.AreaM);

id := 220;	
registry.pointers[id - 1].pFC := ADR(PEU.HysteresisEx);
registry.pointers[id - 1].pB := 0;
registry.pointers[id - 1].vpI._pointer := ADR(GVL.instances.hysteresisEx);
registry.pointers[id - 1].vpI.size := SIZEOF(PEU.HysteresisExInstance);
registry.pointers[id - 1].vpM._pointer := ADR(GVL.m.hysteresisEx);
registry.pointers[id - 1].vpM.size := SIZEOF(PEU.HysteresisExM);
END_METHOD

METHOD PUBLIC initTypes
VAR_INPUT
END_VAR
VAR
	id: UINT;
END_VAR
//TEMPLATE TYPE
FOR id := 1 TO PEC.GC.TEMPLATE_MAX_IDX + 1 DO
	registry.types[id - 1].name := 	'Template';
	registry.types[id - 1].instListName := CONCAT('instances.template[', TO_STRING(id - 1));
	registry.types[id - 1].instListName := CONCAT(registry.types[id - 1].instListName, '].instance');
	registry.types[id - 1]._max := PEC.GC.TEMPLATE_INST_MAX_IDX + 1;
END_FOR;

//INSTRUCTIONS AND SYSTEM CLASSES
id := 150;
registry.types[id - 1].name := 'IEdge';
registry.types[id - 1].instListName := 'instructions.edge';
registry.types[id - 1]._max := GC.IEDGE_M_MAX_IDX + 1;

id := id + 1; //151
registry.types[id - 1].name := 'ITrig';
registry.types[id - 1].instListName := 'instructions.trig';
registry.types[id - 1]._max := GC.ITRIG_M_MAX_IDX + 1;

id := id + 1; //152
registry.types[id - 1].name := 'ITimer';
registry.types[id - 1].instListName := 'instructions.timer';
registry.types[id - 1]._max := GC.ITIMER_MAX_IDX + 1;

id := id + 1; //153
registry.types[id - 1].name := 'ICounter';	
registry.types[id - 1].instListName := 'instructions.counter';
registry.types[id - 1]._max := GC.ICOUNTER_MAX_IDX + 1;

id := id + 1; //154


id := id + 1; //155
registry.types[id - 1].name := 'DigOut';
registry.types[id - 1].instListName := 'instances.digOut';
registry.types[id - 1]._max := GC.DIG_OUT_MAX_IDX + 1;

id := id + 1; //156

id := id + 1; //157
registry.types[id - 1].name := 'DI16';
registry.types[id - 1].instListName := 'hw.di16';
registry.types[id - 1]._max := GC.DI16_MAX_IDX + 1;

id := id + 1; //158
registry.types[id - 1].name := 'DO16';
registry.types[id - 1].instListName := 'hw.do16';
registry.types[id - 1]._max := GC.DO16_MAX_IDX + 1;

id := id + 1; //159
registry.types[id - 1].name := 'AI16';
registry.types[id - 1].instListName := 'hw.ai16';
registry.types[id - 1]._max := GC.AI16_MAX_IDX + 1;

id := id + 1; //160
registry.types[id - 1].name := 'AO4';
registry.types[id - 1].instListName := 'hw.ao4';
registry.types[id - 1]._max := GC.AO4_MAX_IDX + 1;

id := id + 1; //161
registry.types[id - 1].name := 'RcpCommon';
registry.types[id - 1].instListName := 'instructions.rcpCommon';
registry.types[id - 1]._max := PEC.GC.RCP_CALL_INST_MAX_IDX + 1;	

id := id + 1; //162
registry.types[id - 1].name := 'RcpStage';
registry.types[id - 1].instListName := 'instructions.rcpStage';
registry.types[id - 1]._max := PEC.GC.RCP_CALL_INST_MAX_IDX + 1;	

id := id + 1; //163
registry.types[id - 1].name := 'RcpStep';
registry.types[id - 1].instListName := 'instructions.rcpStep';
registry.types[id - 1]._max := PEC.GC.RCP_CALL_INST_MAX_IDX + 1;

id := id + 1; //164
registry.types[id - 1].name := 'Window';
registry.types[id - 1].instListName := 'instances.window';
registry.types[id - 1]._max := PEC.GC.WINDOW_MAX_IDX + 1;

id := id + 1; //165
registry.types[id - 1].name := 'Parameters';
registry.types[id - 1].instListName := 'instances.parameters';
registry.types[id - 1]._max := PEC.GC.PARAMETERS_MAX_IDX + 1;

id := id + 1; //166
registry.types[id - 1].name := 'IPulse';
registry.types[id - 1].instListName := 'instructions.pulse';
registry.types[id - 1]._max := GC.IPULSE_MAX_IDX + 1;

id := id + 1; //167
registry.types[id - 1].name := 'PidC';
registry.types[id - 1].instListName := 'instances.pidC';
registry.types[id - 1]._max := GC.PID_C_MAX_IDX + 1;

//USER TYPES
id := 200;
registry.types[id - 1].name := 'Valve';
registry.types[id - 1].instListName := 'instances.valve';
registry.types[id - 1]._max := GC.VALVE_MAX_IDX + 1;

id := id + 1;
registry.types[id - 1].name := 'ValveReg';
registry.types[id - 1].instListName := 'instances.valveReg';
registry.types[id - 1]._max := GC.VALVE_REG_MAX_IDX + 1;

id := id + 1;
registry.types[id - 1].name := 'Drive';
registry.types[id - 1].instListName := 'instances.drive';
registry.types[id - 1]._max := GC.DRIVE_MAX_IDX + 1;

id := id + 1;
registry.types[id - 1].name := 'DriveReg';
registry.types[id - 1].instListName := 'instances.driveReg';
registry.types[id - 1]._max := GC.DRIVE_REG_MAX_IDX + 1;

id := id + 1;
registry.types[id - 1].name := 'SensorDig';
registry.types[id - 1].instListName := 'instances.sensorDig';
registry.types[id - 1]._max := GC.SENSOR_DIG_MAX_IDX + 1;

id := id + 1;
registry.types[id - 1].name := 'SensorAn';
registry.types[id - 1].instListName := 'instances.sensorAn';
registry.types[id - 1]._max := GC.SENSOR_AN_MAX_IDX + 1;

id := id + 1;

id := id + 1;
registry.types[id - 1].name := 'Hysteresis';
registry.types[id - 1].instListName := 'instances.hysteresis';
registry.types[id - 1]._max := GC.HYSTERESIS_MAX_IDX + 1;

id := id + 1; //208
registry.types[id - 1].name := 'GasFlowReg';
registry.types[id - 1].instListName := 'instances.gasFlowReg';
registry.types[id - 1]._max := GC.GAS_FLOW_REG_MAX_IDX + 1;

id := id + 1; //209
registry.types[id - 1].name := 'Cascade';
registry.types[id - 1].instListName := 'instances.cascade';
registry.types[id - 1]._max := GC.REF_MAX_IDX + 1;

id := id + 1; //210
registry.types[id - 1].name := 'Dose';
registry.types[id - 1].instListName := 'instances.dose';
registry.types[id - 1]._max := GC.DOSE_MAX_IDX + 1;

id := id + 1; //211
registry.types[id - 1].name := 'Profile';
registry.types[id - 1].instListName := 'instances.profile';
registry.types[id - 1]._max := GC.PROFILE_MAX_IDX + 1;

id := id + 1; //212
registry.types[id - 1].name := 'Ramp';
registry.types[id - 1].instListName := 'instances.ramp';
registry.types[id - 1]._max := GC.RAMP_MAX_IDX + 1;	

id := id + 1; //213
registry.types[id - 1].name := 'Route';
registry.types[id - 1].instListName := 'instances.route';
registry.types[id - 1]._max := GC.ROUTE_MAX_IDX + 1;	

id := id + 1; //214
registry.types[id - 1].name := 'Flip';
registry.types[id - 1].instListName := 'instances.flip';
registry.types[id - 1]._max := GC.FLIP_MAX_IDX + 1;

id := id + 1; //215

id := id + 1; //216

id := id + 1; //217

id := id + 1; //218

id := id + 1; //219
registry.types[id - 1].name := 'Area';
registry.types[id - 1].instListName :=  'area';
registry.types[id - 1]._max := GC.AREA_MAX_IDX + 1;

id := id + 1; //220
registry.types[id - 1].name := 'HysteresisEx';
registry.types[id - 1].instListName := 'instances.hysteresisEx';
registry.types[id - 1]._max := GC.HYSTERESISEX_MAX_IDX + 1;
END_METHOD

METHOD PUBLIC updateHW
VAR_INPUT
END_VAR
//GVL.hw.ai16[0].io.error := IoConfig_Globals.NL_S_8AI_16ch_ModBus.xError;
//GVL.hw.di16[0].io.error := IoConfig_Globals.NL_S_16DI_ModBus.xError;
END_METHOD

METHOD exReadTagsCall
VAR_INPUT
END_VAR
VAR
	i: UINT;
	ptr: UDINT;
END_VAR
CASE tagsExM.readState OF
	0: //await new request
		IF(readTagsEx.request.count <> 0) THEN
			tagsExM.readState := 1;
		END_IF;
	1: //update
		FOR i := 0 TO readTagsEx.request.count - 1 DO
			readTagsEx.response.result[i] := checkTagPointer(readTagsEx.request.list[i], ADR(registry));
			IF readTagsEx.response.result[i] > 0 THEN
				CONTINUE;
			END_IF;
			ptr := registry.pointers[readTagsEx.request.list[i].classId - 1].vpI._pointer + 
				registry.pointers[readTagsEx.request.list[i].classId - 1].vpI.size * (readTagsEx.request.list[i].instNum - 1) +
				readTagsEx.request.list[i].offset;				
			MEMUtils.MemCpy(ADR(readTagsEx.response.data[i]), ptr, readTagsEx.request.list[i].size);
		END_FOR
		tagsExM.readState := 2;
	2: //await reset
		IF readTagsEx.request.reset OR tagsExM.readResetTimeout.Q THEN
			MEMUtils.MemSet(ADR(readTagsEx), 0, SIZEOF(readTagsEx));
			tagsExM.readState := 0;
		END_IF
	ELSE
		;
END_CASE

tagsExM.readResetTimeout.IN := tagsExM.readState = 2;
tagsExM.readResetTimeout.PT := T#10S;
tagsExM.readResetTimeout();

readTagsEx.response.busy := tagsExM.readState = 1;
readTagsEx.response.done := tagsExM.readState = 2;
END_METHOD

METHOD exWriteTagsCall
VAR_INPUT
END_VAR
VAR
	i: UINT;
	ptr: UDINT;
END_VAR
CASE tagsExM.writeState OF
	0: //await new request
		IF(writeTagsEx.request.count <> 0) THEN
			tagsExM.writeState := 1;
		END_IF;
	1: //update
		FOR i := 0 TO writeTagsEx.request.count - 1 DO
			writeTagsEx.response.result[i] := checkTagPointer(writeTagsEx.request.list[i], ADR(registry));
			IF writeTagsEx.response.result[i] > 0 THEN
				CONTINUE;
			END_IF;
			ptr := registry.pointers[writeTagsEx.request.list[i].classId - 1].vpI._pointer + 
				registry.pointers[writeTagsEx.request.list[i].classId - 1].vpI.size * (writeTagsEx.request.list[i].instNum - 1) +
				writeTagsEx.request.list[i].offset;
			MEMUtils.MemCpy(ptr, ADR(writeTagsEx.request.data[i]), writeTagsEx.request.list[i].size);
		END_FOR
		tagsExM.writeState := 2;
	2: //await reset
		IF writeTagsEx.request.reset OR tagsExM.writeResetTimeout.Q THEN
			MEMUtils.MemSet(ADR(writeTagsEx), 0, SIZEOF(writeTagsEx));
			tagsExM.writeState := 0;
		END_IF
	ELSE
		;
END_CASE

tagsExM.writeResetTimeout.IN := tagsExM.writeState = 2;
tagsExM.writeResetTimeout.PT := T#10S;
tagsExM.writeResetTimeout();

writeTagsEx.response.busy := tagsExM.writeState = 1;
writeTagsEx.response.done := tagsExM.writeState = 2;
END_METHOD

METHOD templateMonitor
VAR_INPUT
END_VAR
VAR
	status: USINT;
END_VAR
status := PEC.GDBC.dbResultDone;
IF templateMonitorEx.control.enable THEN
	IF templateMonitorEx.control.id = 0 OR templateMonitorEx.control.id > PEC.GC.TEMPLATE_MAX_IDX + 1 THEN
		status := PEC.GDBC.dbResultClassNumError;
	END_IF
	IF templateMonitorEx.control.num = 0 OR templateMonitorEx.control.num > registry.instances[templateMonitorEx.control.id - 1].count THEN
		status := PEC.GDBC.dbResultInstNumError;
	END_IF
	IF templateMonitorEx.control.sum <> registry.instances[templateMonitorEx.control.id - 1].sum THEN
		status := PEC.GDBC.dbResultSumError;
	END_IF
	IF status = PEC.GDBC.dbResultDone THEN
		templateMonitorEx.state.ok := TRUE;
		templateMonitorEx.state.error := FALSE;
	ELSE
		MEMUtils.MemSet(ADR(templateMonitorEx), 0, SIZEOF(templateMonitorEx));
		templateMonitorEx.state.ok := FALSE;
		templateMonitorEx.state.error := TRUE;	
	END_IF
ELSE
	templateMonitorEx.state.ok := FALSE;
	templateMonitorEx.state.error := FALSE;
END_IF
END_METHOD

END_PROGRAM

// A_SIM/PE/MAIN
PROGRAM MAIN
VAR
	callCounter: UINT := 0;
END_VAR
VAR_TEMP
	i: UINT := 0;
END_VAR

IF(GVL.systemData.rt.control.run) THEN
	GVL.systemData.rt.state.mainOff := FALSE;	
	MEMUtils.MemSet(ADR(GVL.systemData.callFlags), 0, SIZEOF(CallFlags));
	GVL.systemData.callFlags.main := TRUE;
	FOR i := 0 TO GC.HCB_MAX_IDX DO
		hcb(ADR(GVL.ex.hcb[i]), ADR(GVL.instances));
	END_FOR;
	PEC.exec(ADR(GVL.systemData));
	FOR i := 0 TO GC.HRB_MAX_IDX DO
		hrb(ADR(GVL.ex.hrb[i]), ADR(GVL.instances));
	END_FOR;
	states(ADR(GVL.ex), ADR(GVL.instances), GVL.systemData.pRegistry);
	GVL.systemData.callFlags.main := FALSE;
	callCounter := callCounter + 1;		
ELSE
	GVL.systemData.rt.state.mainOff := TRUE;	
END_IF;

METHOD PUBLIC hcb
VAR_INPUT
	pHcb: POINTER TO HmiCmdBuffer;
	pI: POINTER TO Instances;
END_VAR
VAR
	n: UINT := 0;
	i: UINT := 0;
END_VAR
IF pHcb^.cLoop.toPlc <> pHcb^.cLoop.fromPlc THEN
	IF pHcb^.count > GC.HC_BUFFER_MAX_IDX + 1 THEN RETURN; END_IF;
	i := 0;
	WHILE i < pHcb^.count DO
		IF(pHcb^.cmd[i].cId = 0 OR pHcb^.cmd[i].iId = 0 OR pHcb^.cmd[i].fc = 0) THEN
			CONTINUE;
		END_IF;
		CASE pHcb^.cmd[i].cId OF
			155: //DIG OUT
				digOutHC(ADR(pI^.digOut[pHcb^.cmd[i].iId - 1]), pHcb^.cmd[i].fc, pHcb^.cmd[i].exId, pHcb^.cmd[i].data);
			164: //WINDOW
				windowHC(ADR(pI^.window[pHcb^.cmd[i].iId - 1]), pHcb^.cmd[i].fc, pHcb^.cmd[i].exId, pHcb^.cmd[i].data);
			165: //PARAMETERS
				parametersHC(ADR(pI^.parameters[pHcb^.cmd[i].iId - 1]), pHcb^.cmd[i].fc, pHcb^.cmd[i].exId, pHcb^.cmd[i].data);
			200: //VALVE
				valveHC(ADR(pI^.valve[pHcb^.cmd[i].iId - 1]), pHcb^.cmd[i].fc, pHcb^.cmd[i].exId, pHcb^.cmd[i].data);
			201: //VALVE REG
				valveRegHC(ADR(pI^.valveReg[pHcb^.cmd[i].iId - 1]), pHcb^.cmd[i].fc, pHcb^.cmd[i].exId, pHcb^.cmd[i].data);
			202: //DRIVE
				driveHC(ADR(pI^.drive[pHcb^.cmd[i].iId - 1]), pHcb^.cmd[i].fc, pHcb^.cmd[i].exId, pHcb^.cmd[i].data);
			203: //DRIVE REG
				driveRegHC(ADR(pI^.driveReg[pHcb^.cmd[i].iId - 1]), pHcb^.cmd[i].fc, pHcb^.cmd[i].exId, pHcb^.cmd[i].data);
			204: //SENSOR DIG
				sensorDigHC(ADR(pI^.sensorDig[pHcb^.cmd[i].iId - 1]), pHcb^.cmd[i].fc, pHcb^.cmd[i].exId, pHcb^.cmd[i].data);
			205: //SENSOR AN
				sensorAnHC(ADR(pI^.sensorAn[pHcb^.cmd[i].iId - 1]), pHcb^.cmd[i].fc, pHcb^.cmd[i].exId, pHcb^.cmd[i].data);
			208: //GAS FLOW REG
				gasFlowRegHC(ADR(pI^.gasFlowReg[pHcb^.cmd[i].iId - 1]), pHcb^.cmd[i].fc, pHcb^.cmd[i].exId, pHcb^.cmd[i].data);			
			ELSE
				;
		END_CASE
		i := i + 1;
	END_WHILE
	
	pHcb^.count := 0;
	MEMUtils.MemSet(ADR(pHcb^.cmd), 0, SIZEOF(pHcb^.cmd));
	pHcb^.cLoop.fromPlc := pHcb^.cLoop.toPlc;
END_IF
END_METHOD

METHOD PUBLIC states
VAR_INPUT
	pEx: POINTER TO Exchange;
	pI : POINTER TO Instances;	
	pR: POINTER TO Registry;
END_VAR
VAR
	n: UINT := 0;
	j: USINT := 0;
	count: UINT := 0;
	bitarray, mask: UDINT;
END_VAR
//WINDOW
count := pR^.instances[164 - 1].count;
n := 1;
WHILE n <= count DO		
	//ERRORS
	bitarray := 0;
	mask := 1;
	FOR j := 0 TO 31 DO
		IF GVL.instances.window[n - 1].plc.error[j] THEN
			bitarray := bitarray OR mask;
		END_IF;
		mask := SHL(mask, 1);
		GVL.instances.window[n - 1].plc.error[j] := 0;
	END_FOR;
	GVL.ex.window.errors[n - 1] := bitarray;
	//LOCKS
	bitarray := 0;
	mask := 1;
	FOR j := 0 TO 31 DO
		IF GVL.instances.window[n - 1].plc.lock[j] THEN
			bitarray := bitarray OR mask;
		END_IF;
		mask := SHL(mask, 1);
		GVL.instances.window[n - 1].plc.lock[j] := 0;
	END_FOR;
	GVL.ex.window.locks[n - 1] := bitarray;
	//OTHER
	MEMUtils.MemCpy(ADR(GVL.ex.window.status[n - 1]), ADR(GVL.instances.window[n - 1].plc.status), 4);
	GVL.instances.window[n - 1].plc.status := 0;
	MEMUtils.MemCpy(ADR(GVL.ex.window.workTime[n - 1]), ADR(GVL.instances.window[n - 1].plc.workTime), 4);
	GVL.instances.window[n - 1].plc.workTime := T#0S;
	//END CODE
	n := n + 1;
END_WHILE;

//VALVE
count :=  pR^.instances[200 - 1].count;
n := 1;
WHILE n <= count DO
	pEx^.valve.status[n - 1] := valveStateToDWord(pI^.valve[n - 1].hmi.state);
	n := n + 1;
END_WHILE;

//VALVE REG
count :=  pR^.instances[201 - 1].count;
n := 1;
WHILE n <= count DO	
	pEx^.valveReg.status[n - 1] := valveRegStateToDWord(pI^.valveReg[n - 1].hmi.state);
	pEx^.valveReg.sp[n - 1] := pI^.valveReg[n - 1].hmi.currentSp;
	n := n + 1;
END_WHILE;

//GAS
count :=  pR^.instances[208 - 1].count;
n := 1;
WHILE n <= count DO
	pEx^.gasFlowReg.status[n - 1] := gasFlowRegStateToDWord(pI^.gasFlowReg[n - 1].hmi.state);
	pEx^.gasFlowReg.sp[n - 1] := pI^.gasFlowReg[n - 1].hmi.currentSp;
	pEx^.gasFlowReg.pv[n - 1] := pI^.gasFlowReg[n - 1].hmi.pv;
	n := n + 1;
END_WHILE;

//DIG OUT
count :=  pR^.instances[155 - 1].count;
n := 1;
WHILE n <= count DO
	pEx^.digOut.status[n - 1] := digOutStateToDWord(pI^.digOut[n - 1].hmi.state);	
	n := n + 1;
END_WHILE;

//DRIVE
count :=  pR^.instances[202 - 1].count;
n := 1;
WHILE n <= count DO
	pEx^.drive.status[n - 1] := driveStateToDWord(pI^.drive[n - 1].hmi.state);
	n := n + 1;
END_WHILE;

//DRIVE REG
count :=  pR^.instances[203 - 1].count;
n := 1;
WHILE n <= count DO
	pEx^.driveReg.status[n - 1] := driveRegStateToDWord(pI^.driveReg[n - 1].hmi.state);
	pEx^.driveReg.sp[n - 1] := pI^.driveReg[n - 1].hmi.currentSp;
	pEx^.driveReg.pv[n - 1] := pI^.driveReg[n - 1].hmi.pv;
	n := n + 1;
END_WHILE;

//SENS DIG
count :=  pR^.instances[204 - 1].count;
n := 1;
WHILE n <= count DO
	pEx^.sensorDig.status[n - 1] := sensorDigStateToDWord(pI^.sensorDig[n - 1].hmi.state);	
	n := n + 1;
END_WHILE;

//SENS AN
count :=  pR^.instances[205 - 1].count;
n := 1;
WHILE n <= count DO
	pEx^.sensorAn.status[n - 1] := sensorAnStateToDWord(pI^.sensorAn[n - 1].hmi.state);
	pEx^.sensorAn.sp[n - 1] := pI^.sensorAn[n - 1].hmi.sp;
	pEx^.sensorAn.pv[n - 1] := pI^.sensorAn[n - 1].hmi.pv;	
	n := n + 1;
END_WHILE;

//PID_C
count :=  pR^.instances[167 - 1].count;
n := 1;
WHILE n <= count DO
	pEx^.pidC.status[n - 1] := pidCStateToDWord(pI^.pidC[n - 1].hmi.state);
	pEx^.pidC.out[n - 1] := pI^.pidC[n - 1].hmi.out;	
	n := n + 1;
END_WHILE;

//HYST
count :=  pR^.instances[207 - 1].count;
n := 1;
WHILE n <= count DO
	pEx^.hysteresis.status[n - 1] := hysteresisStateToDWord(pI^.hysteresis[n - 1].hmi.state);
	pEx^.hysteresis.out1[n - 1] := pI^.hysteresis[n - 1].hmi.out1;
	pEx^.hysteresis.out2[n - 1] := pI^.hysteresis[n - 1].hmi.out2;	
	n := n + 1;
END_WHILE;

//CASCADE
count :=  pR^.instances[209 - 1].count;
n := 1;
WHILE n <= count DO
	pEx^.cascade.status[n - 1] := cascadeStateToDWord(pI^.cascade[n - 1].hmi.state);
	//OUT
	//pEx^.cascade.out[n - 1] := pI^.cascade[n - 1].hmi.out;
	n := n + 1;
END_WHILE;

//HYST EX
count :=  pR^.instances[220 - 1].count;
n := 1;
WHILE n <= count DO
	pEx^.hysteresisEx.status[n - 1] := hysteresisExStateToDWord(pI^.hysteresisEx[n - 1].hmi.state);
	//OUT
	FOR j := 0 TO 4 DO
		pEx^.hysteresisEx.outActuator[n - 1,j] := pI^.hysteresisEx[n - 1].hmi.outActuator[j];
	END_FOR;
	pEx^.hysteresisEx.out[n - 1] := pI^.hysteresisEx[n - 1].hmi.out;
	
	n := n + 1;
END_WHILE;
END_METHOD

METHOD PUBLIC hrb
VAR_INPUT
	pHrb: POINTER TO HmiReadBuffer;
	pI: POINTER TO Instances;
END_VAR
VAR
	n: UINT := 0;
	i: UINT := 0;
END_VAR
IF pHrb^.cLoop.toPlc <> pHrb^.cLoop.fromPlc THEN
	IF pHrb^.count > GC.HR_BUFFER_MAX_IDX + 1 THEN RETURN; END_IF;
	i := 0;
	WHILE i < pHrb^.count DO
		IF(pHrb^.req[i].cId = 0 OR pHrb^.req[i].iId = 0 OR pHrb^.req[i].fc = 0) THEN
			CONTINUE;
		END_IF;
		CASE pHrb^.req[i].cId OF
			155: //DIG OUT
				;//digOutHC(ADR(pI^.digOut[pHrb^.req[i].iId - 1]), pHrb^.req[i].fc, pHrb^.req[i].exId, pHrb^.req[i].data);
			164: //WINDOW
				windowHR(ADR(pI^.window[pHrb^.req[i].iId - 1]), pHrb^.req[i].fc, pHrb^.req[i].exId, pHrb^.res[i].val);
			165: //PARAMETERS
				;//parametersHC(ADR(pI^.parameters[pHrb^.req[i].iId - 1]), pHrb^.req[i].fc, pHrb^.req[i].exId, pHrb^.req[i].data);
			200: //VALVE
				;//valveHC(ADR(pI^.valve[pHrb^.req[i].iId - 1]), pHrb^.req[i].fc, pHrb^.req[i].exId, pHrb^.req[i].data);
			201: //VALVE REG
				;//valveRegHC(ADR(pI^.valveReg[pHrb^.req[i].iId - 1]), pHrb^.req[i].fc, pHrb^.req[i].exId, pHrb^.req[i].data);
			202: //DRIVE
				;//driveHC(ADR(pI^.drive[pHrb^.req[i].iId - 1]), pHrb^.req[i].fc, pHrb^.req[i].exId, pHrb^.req[i].data);
			203: //DRIVE REG
				;//driveRegHC(ADR(pI^.driveReg[pHrb^.req[i].iId - 1]), pHrb^.req[i].fc, pHrb^.req[i].exId, pHrb^.req[i].data);
			204: //SENSOR DIG
				;//sensorDigHC(ADR(pI^.sensorDig[pHrb^.req[i].iId - 1]), pHrb^.req[i].fc, pHrb^.req[i].exId, pHrb^.req[i].data);
			205: //SENSOR AN
				;//sensorAnHC(ADR(pI^.sensorAn[pHrb^.req[i].iId - 1]), pHrb^.req[i].fc, pHrb^.req[i].exId, pHrb^.req[i].data);
			208: //GAS FLOW REG
				;//gasFlowRegHC(ADR(pI^.gasFlowReg[pHrb^.req[i].iId - 1]), pHrb^.req[i].fc, pHrb^.req[i].exId, pHrb^.req[i].data);			
			ELSE
				;
		END_CASE
		i := i + 1;
	END_WHILE
	
	pHrb^.cLoop.fromPlc := pHrb^.cLoop.toPlc;
END_IF
END_METHOD

END_PROGRAM

// RLDA/PE/MAIN
PROGRAM MAIN
VAR
	callCounter: UINT := 0;
END_VAR
VAR_TEMP
	i: UINT := 0;
END_VAR

IF(GVL.systemData.rt.control.run) THEN
	GVL.systemData.rt.state.mainOff := FALSE;	
	MEMUtils.MemSet(ADR(GVL.systemData.callFlags), 0, SIZEOF(CallFlags));
	GVL.systemData.callFlags.main := TRUE;
	FOR i := 0 TO GC.HCB_MAX_IDX DO
		hcb(ADR(GVL.ex.hcb[i]), ADR(GVL.instances));
	END_FOR;
	PEC.exec(ADR(GVL.systemData));
	FOR i := 0 TO GC.HRB_MAX_IDX DO
		hrb(ADR(GVL.ex.hrb[i]), ADR(GVL.instances));
	END_FOR;
	states(ADR(GVL.ex), ADR(GVL.instances), GVL.systemData.pRegistry);
	GVL.systemData.callFlags.main := FALSE;
	callCounter := callCounter + 1;		
ELSE
	GVL.systemData.rt.state.mainOff := TRUE;	
END_IF;

METHOD PUBLIC hcb
VAR_INPUT
	pHcb: POINTER TO HmiCmdBuffer;
	pI: POINTER TO Instances;
END_VAR
VAR
	n: UINT := 0;
	i: UINT := 0;
END_VAR
IF pHcb^.cLoop.toPlc <> pHcb^.cLoop.fromPlc THEN
	IF pHcb^.count > GC.HC_BUFFER_MAX_IDX + 1 THEN RETURN; END_IF;
	i := 0;
	WHILE i < pHcb^.count DO
		IF(pHcb^.cmd[i].cId = 0 OR pHcb^.cmd[i].iId = 0 OR pHcb^.cmd[i].fc = 0) THEN
			CONTINUE;
		END_IF;
		CASE pHcb^.cmd[i].cId OF
			155: //DIG OUT
				digOutHC(ADR(pI^.digOut[pHcb^.cmd[i].iId - 1]), pHcb^.cmd[i].fc, pHcb^.cmd[i].exId, pHcb^.cmd[i].data);
			164: //WINDOW
				windowHC(ADR(pI^.window[pHcb^.cmd[i].iId - 1]), pHcb^.cmd[i].fc, pHcb^.cmd[i].exId, pHcb^.cmd[i].data);
			165: //PARAMETERS
				parametersHC(ADR(pI^.parameters[pHcb^.cmd[i].iId - 1]), pHcb^.cmd[i].fc, pHcb^.cmd[i].exId, pHcb^.cmd[i].data);
			200: //VALVE
				valveHC(ADR(pI^.valve[pHcb^.cmd[i].iId - 1]), pHcb^.cmd[i].fc, pHcb^.cmd[i].exId, pHcb^.cmd[i].data);
			201: //VALVE REG
				valveRegHC(ADR(pI^.valveReg[pHcb^.cmd[i].iId - 1]), pHcb^.cmd[i].fc, pHcb^.cmd[i].exId, pHcb^.cmd[i].data);
			202: //DRIVE
				driveHC(ADR(pI^.drive[pHcb^.cmd[i].iId - 1]), pHcb^.cmd[i].fc, pHcb^.cmd[i].exId, pHcb^.cmd[i].data);
			203: //DRIVE REG
				driveRegHC(ADR(pI^.driveReg[pHcb^.cmd[i].iId - 1]), pHcb^.cmd[i].fc, pHcb^.cmd[i].exId, pHcb^.cmd[i].data);
			204: //SENSOR DIG
				sensorDigHC(ADR(pI^.sensorDig[pHcb^.cmd[i].iId - 1]), pHcb^.cmd[i].fc, pHcb^.cmd[i].exId, pHcb^.cmd[i].data);
			205: //SENSOR AN
				sensorAnHC(ADR(pI^.sensorAn[pHcb^.cmd[i].iId - 1]), pHcb^.cmd[i].fc, pHcb^.cmd[i].exId, pHcb^.cmd[i].data);
			208: //GAS FLOW REG
				gasFlowRegHC(ADR(pI^.gasFlowReg[pHcb^.cmd[i].iId - 1]), pHcb^.cmd[i].fc, pHcb^.cmd[i].exId, pHcb^.cmd[i].data);			
			ELSE
				;
		END_CASE
		i := i + 1;
	END_WHILE
	
	pHcb^.count := 0;
	MEMUtils.MemSet(ADR(pHcb^.cmd), 0, SIZEOF(pHcb^.cmd));
	pHcb^.cLoop.fromPlc := pHcb^.cLoop.toPlc;
END_IF
END_METHOD

METHOD PUBLIC states
VAR_INPUT
	pEx: POINTER TO Exchange;
	pI : POINTER TO Instances;	
	pR: POINTER TO Registry;
END_VAR
VAR
	n: UINT := 0;
	j: USINT := 0;
	count: UINT := 0;
	bitarray, mask: UDINT;
END_VAR
//WINDOW
count := pR^.instances[164 - 1].count;
n := 1;
WHILE n <= count DO		
	//ERRORS
	bitarray := 0;
	mask := 1;
	FOR j := 0 TO 31 DO
		IF GVL.instances.window[n - 1].plc.error[j] THEN
			bitarray := bitarray OR mask;
		END_IF;
		mask := SHL(mask, 1);
		GVL.instances.window[n - 1].plc.error[j] := 0;
	END_FOR;
	GVL.ex.window.errors[n - 1] := bitarray;
	//LOCKS
	bitarray := 0;
	mask := 1;
	FOR j := 0 TO 31 DO
		IF GVL.instances.window[n - 1].plc.lock[j] THEN
			bitarray := bitarray OR mask;
		END_IF;
		mask := SHL(mask, 1);
		GVL.instances.window[n - 1].plc.lock[j] := 0;
	END_FOR;
	GVL.ex.window.locks[n - 1] := bitarray;
	//OTHER
	MEMUtils.MemCpy(ADR(GVL.ex.window.status[n - 1]), ADR(GVL.instances.window[n - 1].plc.status), 4);
	GVL.instances.window[n - 1].plc.status := 0;
	MEMUtils.MemCpy(ADR(GVL.ex.window.workTime[n - 1]), ADR(GVL.instances.window[n - 1].plc.workTime), 4);
	GVL.instances.window[n - 1].plc.workTime := T#0S;
	//END CODE
	n := n + 1;
END_WHILE;

//VALVE
count :=  pR^.instances[200 - 1].count;
n := 1;
WHILE n <= count DO
	pEx^.valve.status[n - 1] := valveStateToDWord(pI^.valve[n - 1].hmi.state);
	n := n + 1;
END_WHILE;

//VALVE REG
count :=  pR^.instances[201 - 1].count;
n := 1;
WHILE n <= count DO	
	pEx^.valveReg.status[n - 1] := valveRegStateToDWord(pI^.valveReg[n - 1].hmi.state);
	pEx^.valveReg.sp[n - 1] := pI^.valveReg[n - 1].hmi.currentSp;
	n := n + 1;
END_WHILE;

//GAS
count :=  pR^.instances[208 - 1].count;
n := 1;
WHILE n <= count DO
	pEx^.gasFlowReg.status[n - 1] := gasFlowRegStateToDWord(pI^.gasFlowReg[n - 1].hmi.state);
	pEx^.gasFlowReg.sp[n - 1] := pI^.gasFlowReg[n - 1].hmi.currentSp;
	pEx^.gasFlowReg.pv[n - 1] := pI^.gasFlowReg[n - 1].hmi.pv;
	n := n + 1;
END_WHILE;

//DIG OUT
count :=  pR^.instances[155 - 1].count;
n := 1;
WHILE n <= count DO
	pEx^.digOut.status[n - 1] := digOutStateToDWord(pI^.digOut[n - 1].hmi.state);	
	n := n + 1;
END_WHILE;

//DRIVE
count :=  pR^.instances[202 - 1].count;
n := 1;
WHILE n <= count DO
	pEx^.drive.status[n - 1] := driveStateToDWord(pI^.drive[n - 1].hmi.state);
	n := n + 1;
END_WHILE;

//DRIVE REG
count :=  pR^.instances[203 - 1].count;
n := 1;
WHILE n <= count DO
	pEx^.driveReg.status[n - 1] := driveRegStateToDWord(pI^.driveReg[n - 1].hmi.state);
	pEx^.driveReg.sp[n - 1] := pI^.driveReg[n - 1].hmi.currentSp;
	pEx^.driveReg.pv[n - 1] := pI^.driveReg[n - 1].hmi.pv;
	n := n + 1;
END_WHILE;

//SENS DIG
count :=  pR^.instances[204 - 1].count;
n := 1;
WHILE n <= count DO
	pEx^.sensorDig.status[n - 1] := sensorDigStateToDWord(pI^.sensorDig[n - 1].hmi.state);	
	n := n + 1;
END_WHILE;

//SENS AN
count :=  pR^.instances[205 - 1].count;
n := 1;
WHILE n <= count DO
	pEx^.sensorAn.status[n - 1] := sensorAnStateToDWord(pI^.sensorAn[n - 1].hmi.state);
	pEx^.sensorAn.sp[n - 1] := pI^.sensorAn[n - 1].hmi.sp;
	pEx^.sensorAn.pv[n - 1] := pI^.sensorAn[n - 1].hmi.pv;	
	n := n + 1;
END_WHILE;

//PID_C
count :=  pR^.instances[167 - 1].count;
n := 1;
WHILE n <= count DO
	pEx^.pidC.status[n - 1] := pidCStateToDWord(pI^.pidC[n - 1].hmi.state);
	pEx^.pidC.out[n - 1] := pI^.pidC[n - 1].hmi.out;	
	n := n + 1;
END_WHILE;

//HYST
count :=  pR^.instances[207 - 1].count;
n := 1;
WHILE n <= count DO
	pEx^.hysteresis.status[n - 1] := hysteresisStateToDWord(pI^.hysteresis[n - 1].hmi.state);
	pEx^.hysteresis.out1[n - 1] := pI^.hysteresis[n - 1].hmi.out1;
	pEx^.hysteresis.out2[n - 1] := pI^.hysteresis[n - 1].hmi.out2;	
	n := n + 1;
END_WHILE;

//CASCADE
count :=  pR^.instances[209 - 1].count;
n := 1;
WHILE n <= count DO
	pEx^.cascade.status[n - 1] := cascadeStateToDWord(pI^.cascade[n - 1].hmi.state);
	//OUT
	//pEx^.cascade.out[n - 1] := pI^.cascade[n - 1].hmi.out;
	n := n + 1;
END_WHILE;

//HYST EX
count :=  pR^.instances[220 - 1].count;
n := 1;
WHILE n <= count DO
	pEx^.hysteresisEx.status[n - 1] := hysteresisExStateToDWord(pI^.hysteresisEx[n - 1].hmi.state);
	//OUT
	FOR j := 0 TO 4 DO
		pEx^.hysteresisEx.outActuator[n - 1,j] := pI^.hysteresisEx[n - 1].hmi.outActuator[j];
	END_FOR;
	pEx^.hysteresisEx.out[n - 1] := pI^.hysteresisEx[n - 1].hmi.out;
	
	n := n + 1;
END_WHILE;
END_METHOD

METHOD PUBLIC hrb
VAR_INPUT
	pHrb: POINTER TO HmiReadBuffer;
	pI: POINTER TO Instances;
END_VAR
VAR
	n: UINT := 0;
	i: UINT := 0;
END_VAR
IF pHrb^.cLoop.toPlc <> pHrb^.cLoop.fromPlc THEN
	IF pHrb^.count > GC.HR_BUFFER_MAX_IDX + 1 THEN RETURN; END_IF;
	i := 0;
	WHILE i < pHrb^.count DO
		IF(pHrb^.req[i].cId = 0 OR pHrb^.req[i].iId = 0 OR pHrb^.req[i].fc = 0) THEN
			CONTINUE;
		END_IF;
		CASE pHrb^.req[i].cId OF
			155: //DIG OUT
				;//digOutHC(ADR(pI^.digOut[pHrb^.req[i].iId - 1]), pHrb^.req[i].fc, pHrb^.req[i].exId, pHrb^.req[i].data);
			164: //WINDOW
				windowHR(ADR(pI^.window[pHrb^.req[i].iId - 1]), pHrb^.req[i].fc, pHrb^.req[i].exId, pHrb^.res[i].val);
			165: //PARAMETERS
				;//parametersHC(ADR(pI^.parameters[pHrb^.req[i].iId - 1]), pHrb^.req[i].fc, pHrb^.req[i].exId, pHrb^.req[i].data);
			200: //VALVE
				;//valveHC(ADR(pI^.valve[pHrb^.req[i].iId - 1]), pHrb^.req[i].fc, pHrb^.req[i].exId, pHrb^.req[i].data);
			201: //VALVE REG
				;//valveRegHC(ADR(pI^.valveReg[pHrb^.req[i].iId - 1]), pHrb^.req[i].fc, pHrb^.req[i].exId, pHrb^.req[i].data);
			202: //DRIVE
				;//driveHC(ADR(pI^.drive[pHrb^.req[i].iId - 1]), pHrb^.req[i].fc, pHrb^.req[i].exId, pHrb^.req[i].data);
			203: //DRIVE REG
				;//driveRegHC(ADR(pI^.driveReg[pHrb^.req[i].iId - 1]), pHrb^.req[i].fc, pHrb^.req[i].exId, pHrb^.req[i].data);
			204: //SENSOR DIG
				;//sensorDigHC(ADR(pI^.sensorDig[pHrb^.req[i].iId - 1]), pHrb^.req[i].fc, pHrb^.req[i].exId, pHrb^.req[i].data);
			205: //SENSOR AN
				;//sensorAnHC(ADR(pI^.sensorAn[pHrb^.req[i].iId - 1]), pHrb^.req[i].fc, pHrb^.req[i].exId, pHrb^.req[i].data);
			208: //GAS FLOW REG
				;//gasFlowRegHC(ADR(pI^.gasFlowReg[pHrb^.req[i].iId - 1]), pHrb^.req[i].fc, pHrb^.req[i].exId, pHrb^.req[i].data);			
			ELSE
				;
		END_CASE
		i := i + 1;
	END_WHILE
	
	pHrb^.cLoop.fromPlc := pHrb^.cLoop.toPlc;
END_IF
END_METHOD

END_PROGRAM

// RLDA/PE/SYS
PROGRAM SYS
VAR	
	registry: PEC.Registry;
	templateMonitorEx : TemplateMonitorEx;
	id: UINT;
	descriptions: Descriptions;
	readTagsEx: PEC.ReadTagsEx;
	writeTagsEx: PEC.WriteTagsEx;	
	xInit: BOOL := TRUE;
	xReq: BOOL := FALSE;
	tagsExM: TagsExM;
	persistList: PersistList;
END_VAR

GVL.systemData.xFalse := FALSE;
GVL.systemData.xTrue := TRUE;
GVL.systemData.db.control.enable := TRUE;
GVL.systemData.rt.control.run := GVL.systemData.db.state.run;

initTypes();
updatePointers();
exReadTagsCall();
exWriteTagsCall();
templateMonitor();

(*IF GVL.systemData.db.state.run THEN 
	updateHW();	
	
	id := 158;
	registry.instances[id - 1].count := 1;
	registry.instances[id - 1].name := 'DO16';
	registry.instances[id - 1].flags.main := TRUE;
	registry.instances[id - 1].sum := 629;
	
	id := 159;
	registry.instances[id - 1].count := 1;
	registry.instances[id - 1].name := 'AI16';
	registry.instances[id - 1].flags.main := TRUE;
	registry.instances[id - 1].sum := 659;
	
	id := 200;
	registry.instances[id - 1].count := 5;
	registry.instances[id - 1].name := 'Valve';
	registry.instances[id - 1].flags.main := TRUE;
	registry.instances[id - 1].sum := 7287;	
END_IF*)

METHOD PUBLIC updateHW
VAR_INPUT
END_VAR
//GVL.hw.ai16[0].io.error := IoConfig_Globals.NL_S_8AI_16ch_ModBus.xError;
//GVL.hw.di16[0].io.error := IoConfig_Globals.NL_S_16DI_ModBus.xError;
END_METHOD

METHOD PUBLIC updatePointers
VAR_INPUT
END_VAR
VAR
	id: UINT;
END_VAR
//SYSTEM DATA
GVL.systemData.pStack := 0;
GVL.systemData.pRegistry := ADR(SYS.registry);
GVL.systemData.pRecipes := 0;
GVL.systemData.pTemplates := ADR(GVL.templates);
GVL.systemData.pInterfaces := ADR(GVL.interfaces);
GVL.systemData.pTemplateMonitorEx := ADR(templateMonitorEx);
GVL.systemData.pAcc := 0;
GVL.systemData.pSlaves := 0;
GVL.systemData.pPersistList := ADR(persistList);

FOR id := 1 TO PEC.GC.TEMPLATE_MAX_IDX + 1 DO
		registry.pointers[id - 1].pFC := ADR(Template);
		registry.pointers[id - 1].pB := ADR(GVL.templates[id - 1]);
		registry.pointers[id - 1].vpI._pointer := ADR(GVL.instances.template[id - 1]);
		registry.pointers[id - 1].vpI.size := SIZEOF(TemplateInstance);
		registry.pointers[id - 1].vpM._pointer := ADR(GVL.m.template[id - 1]);
		registry.pointers[id - 1].vpM.size := SIZEOF(TemplateInstM);
END_FOR

//INSTRUCTIONS AND SYSTEM CLASSES
id := 150;	//IEdge
registry.pointers[id - 1].pFC := ADR(PEC.IEdge);
registry.pointers[id - 1].pB := 0;
registry.pointers[id - 1].vpI._pointer := ADR(GVL.instructions.edge);
registry.pointers[id - 1].vpI.size := SIZEOF(PEC.IEdgeInstance);
registry.pointers[id - 1].vpM._pointer := 0;
registry.pointers[id - 1].vpM.size := 0;

id := 151; //ITrig
registry.pointers[id - 1].pFC := ADR(PEC.ITrig);
registry.pointers[id - 1].pB := 0;
registry.pointers[id - 1].vpI._pointer := ADR(GVL.instructions.trig);
registry.pointers[id - 1].vpI.size := SIZEOF(PEC.ITrigInstance);
registry.pointers[id - 1].vpM._pointer := 0;
registry.pointers[id - 1].vpM.size := 0;

id := 152; //ITimer
registry.pointers[id - 1].pFC := ADR(PEC.ITimer);
registry.pointers[id - 1].pB := 0;
registry.pointers[id - 1].vpI._pointer := ADR(GVL.instructions.timer);
registry.pointers[id - 1].vpI.size := SIZEOF(PEC.ITimerInstance);
registry.pointers[id - 1].vpM._pointer := 0;
registry.pointers[id - 1].vpM.size := 0;

id := 153; //ICounter
registry.pointers[id - 1].pFC := ADR(PEC.ICounter);
registry.pointers[id - 1].pB := 0;
registry.pointers[id - 1].vpI._pointer := ADR(GVL.instructions.counter);
registry.pointers[id - 1].vpI.size := SIZEOF(PEC.ICounterInstance);
registry.pointers[id - 1].vpM._pointer := 0;
registry.pointers[id - 1].vpM.size := 0;

id := 155; //DigOut
registry.pointers[id - 1].pFC := ADR(PEU.DigOut);
registry.pointers[id - 1].pB := 0;
registry.pointers[id - 1].vpI._pointer := ADR(GVL.instances.digOut);
registry.pointers[id - 1].vpI.size := SIZEOF(PEU.DigOutInstance);
registry.pointers[id - 1].vpM._pointer := ADR(GVL.m.digOut);;
registry.pointers[id - 1].vpM.size := SIZEOF(PEU.digOutM);

id := 157; //DI16
registry.pointers[id - 1].pFC := ADR(PEU.DI16);
registry.pointers[id - 1].pB := 0;
registry.pointers[id - 1].vpI._pointer := ADR(GVL.hw.di16);
registry.pointers[id - 1].vpI.size := SIZEOF(PEU.DI16Instance);
registry.pointers[id - 1].vpM._pointer := ADR(GVL.m.di16);;
registry.pointers[id - 1].vpM.size := SIZEOF(PEU.DI16M);

id := 158; //DO16
registry.pointers[id - 1].pFC := ADR(PEU.DO16);
registry.pointers[id - 1].pB := 0;
registry.pointers[id - 1].vpI._pointer := ADR(GVL.hw.do16);
registry.pointers[id - 1].vpI.size := SIZEOF(PEU.DO16Instance);
registry.pointers[id - 1].vpM._pointer := ADR(GVL.m.do16);;
registry.pointers[id - 1].vpM.size := SIZEOF(PEU.DO16M);

id := 159; //AI16
registry.pointers[id - 1].pFC := ADR(PEU.AI16);
registry.pointers[id - 1].pB := 0;
registry.pointers[id - 1].vpI._pointer := ADR(GVL.hw.ai16);
registry.pointers[id - 1].vpI.size := SIZEOF(PEU.AI16Instance);
registry.pointers[id - 1].vpM._pointer := ADR(GVL.m.ai16);;
registry.pointers[id - 1].vpM.size := SIZEOF(PEU.AI16M);

id := 160; //AO4
registry.pointers[id - 1].pFC := ADR(PEU.AO4);
registry.pointers[id - 1].pB := 0;
registry.pointers[id - 1].vpI._pointer := ADR(GVL.hw.ao4);
registry.pointers[id - 1].vpI.size := SIZEOF(PEU.AO4Instance);
registry.pointers[id - 1].vpM._pointer := ADR(GVL.m.ao4);;
registry.pointers[id - 1].vpM.size := SIZEOF(PEU.AO4M);


id := 161; //RcpCommon	
registry.pointers[id - 1].pFC := ADR(PEC.RcpCommon);
registry.pointers[id - 1].pB := 0;
registry.pointers[id - 1].vpI._pointer := ADR(GVL.instructions.rcpCommon);
registry.pointers[id - 1].vpI.size := SIZEOF(PEC.RcpCommonInstance);
registry.pointers[id - 1].vpM._pointer := ADR(GVL.m.rcpCommon);
registry.pointers[id - 1].vpM.size := SIZEOF(PEC.RcpCommonM);

id := 162; //RcpStage
registry.pointers[id - 1].pFC := ADR(PEC.RcpStage);
registry.pointers[id - 1].pB := 0;
registry.pointers[id - 1].vpI._pointer := ADR(GVL.instructions.rcpStage);
registry.pointers[id - 1].vpI.size := SIZEOF(PEC.RcpStageInstance);
registry.pointers[id - 1].vpM._pointer := ADR(GVL.m.rcpStage);
registry.pointers[id - 1].vpM.size := SIZEOF(PEC.RcpStageM);

id := 163; //RcpStep
registry.pointers[id - 1].pFC := ADR(PEC.RcpStep);
registry.pointers[id - 1].pB := 0;
registry.pointers[id - 1].vpI._pointer := ADR(GVL.instructions.rcpStep);
registry.pointers[id - 1].vpI.size := SIZEOF(PEC.RcpStepInstance);
registry.pointers[id - 1].vpM._pointer := ADR(GVL.m.rcpStep);
registry.pointers[id - 1].vpM.size := SIZEOF(PEC.RcpStepM);

id := 164; //Window
registry.pointers[id - 1].pFC := ADR(PEC.Window);
registry.pointers[id - 1].pB := 0;
registry.pointers[id - 1].vpI._pointer := ADR(GVL.instances.window);
registry.pointers[id - 1].vpI.size := SIZEOF(PEC.WindowInstance);
registry.pointers[id - 1].vpM._pointer := ADR(GVL.m.window);
registry.pointers[id - 1].vpM.size := SIZEOF(PEC.WindowM);

id := 165; //Parameters
registry.pointers[id - 1].pFC := ADR(PEC.Parameters);
registry.pointers[id - 1].pB := 0;
registry.pointers[id - 1].vpI._pointer := ADR(GVL.instances.parameters);
registry.pointers[id - 1].vpI.size := SIZEOF(PEC.ParametersInstance);
registry.pointers[id - 1].vpM._pointer := ADR(GVL.m.parameters);
registry.pointers[id - 1].vpM.size := SIZEOF(PEC.ParametersM);

id := 166; //IPulse
registry.pointers[id - 1].pFC := ADR(PEC.IPulse);
registry.pointers[id - 1].pB := 0;
registry.pointers[id - 1].vpI._pointer := ADR(GVL.instructions.pulse);
registry.pointers[id - 1].vpI.size := SIZEOF(PEC.IPulseInstance);
registry.pointers[id - 1].vpM._pointer := 0;
registry.pointers[id - 1].vpM.size := 0;

//USER TYPES
id := 200;	
registry.pointers[id - 1].pFC := ADR(PEU.Valve);
registry.pointers[id - 1].pB := 0;
registry.pointers[id - 1].vpI._pointer := ADR(GVL.instances.valve);
registry.pointers[id - 1].vpI.size := SIZEOF(PEU.ValveInstance);
registry.pointers[id - 1].vpM._pointer := ADR(GVL.m.valve);
registry.pointers[id - 1].vpM.size := SIZEOF(PEU.ValveM);

id := 201;	
registry.pointers[id - 1].pFC := ADR(PEU.ValveReg);
registry.pointers[id - 1].pB := 0;
registry.pointers[id - 1].vpI._pointer := ADR(GVL.instances.valveReg);
registry.pointers[id - 1].vpI.size := SIZEOF(PEU.ValveRegInstance);
registry.pointers[id - 1].vpM._pointer := ADR(GVL.m.valveReg);
registry.pointers[id - 1].vpM.size := SIZEOF(PEU.ValveRegM);

id := 202;	
registry.pointers[id - 1].pFC := ADR(PEU.Drive);
registry.pointers[id - 1].pB := 0;
registry.pointers[id - 1].vpI._pointer := ADR(GVL.instances.drive);
registry.pointers[id - 1].vpI.size := SIZEOF(PEU.DriveInstance);
registry.pointers[id - 1].vpM._pointer := ADR(GVL.m.drive);
registry.pointers[id - 1].vpM.size := SIZEOF(PEU.DriveM);

id := 203;	
registry.pointers[id - 1].pFC := ADR(PEU.DriveReg);
registry.pointers[id - 1].pB := 0;
registry.pointers[id - 1].vpI._pointer := ADR(GVL.instances.driveReg);
registry.pointers[id - 1].vpI.size := SIZEOF(PEU.DriveRegInstance);
registry.pointers[id - 1].vpM._pointer := ADR(GVL.m.driveReg);
registry.pointers[id - 1].vpM.size := SIZEOF(PEU.DriveRegM);

id := 204;	
registry.pointers[id - 1].pFC := ADR(PEU.SensorDig);
registry.pointers[id - 1].pB := 0;
registry.pointers[id - 1].vpI._pointer := ADR(GVL.instances.sensorDig);
registry.pointers[id - 1].vpI.size := SIZEOF(PEU.SensorDigInstance);
registry.pointers[id - 1].vpM._pointer := ADR(GVL.m.sensorDig);
registry.pointers[id - 1].vpM.size := SIZEOF(PEU.SensorDigM);

id := 205;	
registry.pointers[id - 1].pFC := ADR(PEU.SensorAn);
registry.pointers[id - 1].pB := 0;
registry.pointers[id - 1].vpI._pointer := ADR(GVL.instances.sensorAn);
registry.pointers[id - 1].vpI.size := SIZEOF(PEU.SensorAnInstance);
registry.pointers[id - 1].vpM._pointer := ADR(GVL.m.sensorAn);
registry.pointers[id - 1].vpM.size := SIZEOF(PEU.SensorAnM);

id := 206;


id := 207;	
registry.pointers[id - 1].pFC := ADR(PEU.Hysteresis);
registry.pointers[id - 1].pB := 0;
registry.pointers[id - 1].vpI._pointer := ADR(GVL.instances.hysteresis);
registry.pointers[id - 1].vpI.size := SIZEOF(PEU.HysteresisInstance);
registry.pointers[id - 1].vpM._pointer := ADR(GVL.m.hysteresis);
registry.pointers[id - 1].vpM.size := SIZEOF(PEU.HysteresisM);

id := 208;	
registry.pointers[id - 1].pFC := ADR(PEU.GasFlowReg);
registry.pointers[id - 1].pB := 0;
registry.pointers[id - 1].vpI._pointer := ADR(GVL.instances.gasFlowReg);
registry.pointers[id - 1].vpI.size := SIZEOF(PEU.GasFlowRegInstance);
registry.pointers[id - 1].vpM._pointer := ADR(GVL.m.gasFlowReg);
registry.pointers[id - 1].vpM.size := SIZEOF(PEU.GasFlowRegM);

id := 209;	
registry.pointers[id - 1].pFC := ADR(PEU.Cascade);
registry.pointers[id - 1].pB := 0;
registry.pointers[id - 1].vpI._pointer := ADR(GVL.instances.cascade);
registry.pointers[id - 1].vpI.size := SIZEOF(PEU.CascadeInstance);
registry.pointers[id - 1].vpM._pointer := ADR(GVL.m.cascade);
registry.pointers[id - 1].vpM.size := SIZEOF(PEU.CascadeM);

id := 210;	
registry.pointers[id - 1].pFC := ADR(PEU.Dose);
registry.pointers[id - 1].pB := 0;
registry.pointers[id - 1].vpI._pointer := ADR(GVL.instances.dose);
registry.pointers[id - 1].vpI.size := SIZEOF(PEU.DoseInstance);
registry.pointers[id - 1].vpM._pointer := ADR(GVL.m.dose);
registry.pointers[id - 1].vpM.size := SIZEOF(PEU.DoseM);

id := 211;	
registry.pointers[id - 1].pFC := ADR(PEU.Profile);
registry.pointers[id - 1].pB := 0;
registry.pointers[id - 1].vpI._pointer := ADR(GVL.instances.profile);
registry.pointers[id - 1].vpI.size := SIZEOF(PEU.ProfileInstance);
registry.pointers[id - 1].vpM._pointer := ADR(GVL.m.profile);
registry.pointers[id - 1].vpM.size := SIZEOF(PEU.ProfileM);

id := 212;	
registry.pointers[id - 1].pFC := ADR(PEU.Ramp);
registry.pointers[id - 1].pB := 0;
registry.pointers[id - 1].vpI._pointer := ADR(GVL.instances.ramp);
registry.pointers[id - 1].vpI.size := SIZEOF(PEU.RampInstance);
registry.pointers[id - 1].vpM._pointer := ADR(GVL.m.ramp);
registry.pointers[id - 1].vpM.size := SIZEOF(PEU.RampM);

id := 213;	
registry.pointers[id - 1].pFC := ADR(PEU.Route);
registry.pointers[id - 1].pB := 0;
registry.pointers[id - 1].vpI._pointer := ADR(GVL.instances.route);
registry.pointers[id - 1].vpI.size := SIZEOF(PEU.RouteInstance);
registry.pointers[id - 1].vpM._pointer := ADR(GVL.m.route);
registry.pointers[id - 1].vpM.size := SIZEOF(PEU.RouteM);

id := 214;	
registry.pointers[id - 1].pFC := ADR(PEU.Flip);
registry.pointers[id - 1].pB := 0;
registry.pointers[id - 1].vpI._pointer := ADR(GVL.instances.flip);
registry.pointers[id - 1].vpI.size := SIZEOF(PEU.FlipInstance);
registry.pointers[id - 1].vpM._pointer := ADR(GVL.m.flip);
registry.pointers[id - 1].vpM.size := SIZEOF(PEU.FlipM);

id := 219;	
registry.pointers[id - 1].pFC := ADR(PEU.Area);
registry.pointers[id - 1].pB := 0;
registry.pointers[id - 1].vpI._pointer := ADR(GVL.area);
registry.pointers[id - 1].vpI.size := SIZEOF(PEU.AreaInstance);
registry.pointers[id - 1].vpM._pointer := ADR(GVL.m.area);
registry.pointers[id - 1].vpM.size := SIZEOF(PEU.AreaM);

id := 220;	
registry.pointers[id - 1].pFC := ADR(PEU.HysteresisEx);
registry.pointers[id - 1].pB := 0;
registry.pointers[id - 1].vpI._pointer := ADR(GVL.instances.hysteresisEx);
registry.pointers[id - 1].vpI.size := SIZEOF(PEU.HysteresisExInstance);
registry.pointers[id - 1].vpM._pointer := ADR(GVL.m.hysteresisEx);
registry.pointers[id - 1].vpM.size := SIZEOF(PEU.HysteresisExM);
END_METHOD

METHOD exReadTagsCall
VAR_INPUT
END_VAR
VAR
	i: UINT;
	ptr: UDINT;
END_VAR
CASE tagsExM.readState OF
	0: //await new request
		IF(readTagsEx.request.count <> 0) THEN
			tagsExM.readState := 1;
		END_IF;
	1: //update
		FOR i := 0 TO readTagsEx.request.count - 1 DO
			readTagsEx.response.result[i] := checkTagPointer(readTagsEx.request.list[i], ADR(registry));
			IF readTagsEx.response.result[i] > 0 THEN
				CONTINUE;
			END_IF;
			ptr := registry.pointers[readTagsEx.request.list[i].classId - 1].vpI._pointer + 
				registry.pointers[readTagsEx.request.list[i].classId - 1].vpI.size * (readTagsEx.request.list[i].instNum - 1) +
				readTagsEx.request.list[i].offset;				
			MEMUtils.MemCpy(ADR(readTagsEx.response.data[i]), ptr, readTagsEx.request.list[i].size);
		END_FOR
		tagsExM.readState := 2;
	2: //await reset
		IF readTagsEx.request.reset OR tagsExM.readResetTimeout.Q THEN
			MEMUtils.MemSet(ADR(readTagsEx), 0, SIZEOF(readTagsEx));
			tagsExM.readState := 0;
		END_IF
	ELSE
		;
END_CASE

tagsExM.readResetTimeout.IN := tagsExM.readState = 2;
tagsExM.readResetTimeout.PT := T#10S;
tagsExM.readResetTimeout();

readTagsEx.response.busy := tagsExM.readState = 1;
readTagsEx.response.done := tagsExM.readState = 2;
END_METHOD

METHOD exWriteTagsCall
VAR_INPUT
END_VAR
VAR
	i: UINT;
	ptr: UDINT;
END_VAR
CASE tagsExM.writeState OF
	0: //await new request
		IF(writeTagsEx.request.count <> 0) THEN
			tagsExM.writeState := 1;
		END_IF;
	1: //update
		FOR i := 0 TO writeTagsEx.request.count - 1 DO
			writeTagsEx.response.result[i] := checkTagPointer(writeTagsEx.request.list[i], ADR(registry));
			IF writeTagsEx.response.result[i] > 0 THEN
				CONTINUE;
			END_IF;
			ptr := registry.pointers[writeTagsEx.request.list[i].classId - 1].vpI._pointer + 
				registry.pointers[writeTagsEx.request.list[i].classId - 1].vpI.size * (writeTagsEx.request.list[i].instNum - 1) +
				writeTagsEx.request.list[i].offset;
			MEMUtils.MemCpy(ptr, ADR(writeTagsEx.request.data[i]), writeTagsEx.request.list[i].size);
		END_FOR
		tagsExM.writeState := 2;
	2: //await reset
		IF writeTagsEx.request.reset OR tagsExM.writeResetTimeout.Q THEN
			MEMUtils.MemSet(ADR(writeTagsEx), 0, SIZEOF(writeTagsEx));
			tagsExM.writeState := 0;
		END_IF
	ELSE
		;
END_CASE

tagsExM.writeResetTimeout.IN := tagsExM.writeState = 2;
tagsExM.writeResetTimeout.PT := T#10S;
tagsExM.writeResetTimeout();

writeTagsEx.response.busy := tagsExM.writeState = 1;
writeTagsEx.response.done := tagsExM.writeState = 2;
END_METHOD

METHOD templateMonitor
VAR_INPUT
END_VAR
VAR
	status: USINT;
END_VAR
status := PEC.GDBC.dbResultDone;
IF templateMonitorEx.control.enable THEN
	IF templateMonitorEx.control.id = 0 OR templateMonitorEx.control.id > PEC.GC.TEMPLATE_MAX_IDX + 1 THEN
		status := PEC.GDBC.dbResultClassNumError;
	END_IF
	IF templateMonitorEx.control.num = 0 OR templateMonitorEx.control.num > registry.instances[templateMonitorEx.control.id - 1].count THEN
		status := PEC.GDBC.dbResultInstNumError;
	END_IF
	IF templateMonitorEx.control.sum <> registry.instances[templateMonitorEx.control.id - 1].sum THEN
		status := PEC.GDBC.dbResultSumError;
	END_IF
	IF status = PEC.GDBC.dbResultDone THEN
		templateMonitorEx.state.ok := TRUE;
		templateMonitorEx.state.error := FALSE;
	ELSE
		MEMUtils.MemSet(ADR(templateMonitorEx), 0, SIZEOF(templateMonitorEx));
		templateMonitorEx.state.ok := FALSE;
		templateMonitorEx.state.error := TRUE;	
	END_IF
ELSE
	templateMonitorEx.state.ok := FALSE;
	templateMonitorEx.state.error := FALSE;
END_IF
END_METHOD

METHOD PUBLIC initTypes
VAR_INPUT
END_VAR
VAR
	id: UINT;
END_VAR
//TEMPLATE TYPE
FOR id := 1 TO PEC.GC.TEMPLATE_MAX_IDX + 1 DO
	registry.types[id - 1].name := 	'Template';
	registry.types[id - 1].instListName := CONCAT('instances.template[', TO_STRING(id - 1));
	registry.types[id - 1].instListName := CONCAT(registry.types[id - 1].instListName, '].instance');
	registry.types[id - 1]._max := PEC.GC.TEMPLATE_INST_MAX_IDX + 1;
END_FOR;

//INSTRUCTIONS AND SYSTEM CLASSES
id := 150;
registry.types[id - 1].name := 'IEdge';
registry.types[id - 1].instListName := 'instructions.edge';
registry.types[id - 1]._max := GC.IEDGE_M_MAX_IDX + 1;

id := id + 1; //151
registry.types[id - 1].name := 'ITrig';
registry.types[id - 1].instListName := 'instructions.trig';
registry.types[id - 1]._max := GC.ITRIG_M_MAX_IDX + 1;

id := id + 1; //152
registry.types[id - 1].name := 'ITimer';
registry.types[id - 1].instListName := 'instructions.timer';
registry.types[id - 1]._max := GC.ITIMER_MAX_IDX + 1;

id := id + 1; //153
registry.types[id - 1].name := 'ICounter';	
registry.types[id - 1].instListName := 'instructions.counter';
registry.types[id - 1]._max := GC.ICOUNTER_MAX_IDX + 1;

id := id + 1; //154


id := id + 1; //155
registry.types[id - 1].name := 'DigOut';
registry.types[id - 1].instListName := 'instances.digOut';
registry.types[id - 1]._max := GC.DIG_OUT_MAX_IDX + 1;

id := id + 1; //156

id := id + 1; //157
registry.types[id - 1].name := 'DI16';
registry.types[id - 1].instListName := 'hw.di16';
registry.types[id - 1]._max := GC.DI16_MAX_IDX + 1;

id := id + 1; //158
registry.types[id - 1].name := 'DO16';
registry.types[id - 1].instListName := 'hw.do16';
registry.types[id - 1]._max := GC.DO16_MAX_IDX + 1;

id := id + 1; //159
registry.types[id - 1].name := 'AI16';
registry.types[id - 1].instListName := 'hw.ai16';
registry.types[id - 1]._max := GC.AI16_MAX_IDX + 1;

id := id + 1; //160
registry.types[id - 1].name := 'AO4';
registry.types[id - 1].instListName := 'hw.ao4';
registry.types[id - 1]._max := GC.AO4_MAX_IDX + 1;

id := id + 1; //161
registry.types[id - 1].name := 'RcpCommon';
registry.types[id - 1].instListName := 'instructions.rcpCommon';
registry.types[id - 1]._max := PEC.GC.RCP_CALL_INST_MAX_IDX + 1;	

id := id + 1; //162
registry.types[id - 1].name := 'RcpStage';
registry.types[id - 1].instListName := 'instructions.rcpStage';
registry.types[id - 1]._max := PEC.GC.RCP_CALL_INST_MAX_IDX + 1;	

id := id + 1; //163
registry.types[id - 1].name := 'RcpStep';
registry.types[id - 1].instListName := 'instructions.rcpStep';
registry.types[id - 1]._max := PEC.GC.RCP_CALL_INST_MAX_IDX + 1;

id := id + 1; //164
registry.types[id - 1].name := 'Window';
registry.types[id - 1].instListName := 'instances.window';
registry.types[id - 1]._max := PEC.GC.WINDOW_MAX_IDX + 1;

id := id + 1; //165
registry.types[id - 1].name := 'Parameters';
registry.types[id - 1].instListName := 'instances.parameters';
registry.types[id - 1]._max := PEC.GC.PARAMETERS_MAX_IDX + 1;

id := id + 1; //166
registry.types[id - 1].name := 'IPulse';
registry.types[id - 1].instListName := 'instructions.pulse';
registry.types[id - 1]._max := GC.IPULSE_MAX_IDX + 1;

id := id + 1; //167
registry.types[id - 1].name := 'PidC';
registry.types[id - 1].instListName := 'instances.pidC';
registry.types[id - 1]._max := GC.PID_C_MAX_IDX + 1;

//USER TYPES
id := 200;
registry.types[id - 1].name := 'Valve';
registry.types[id - 1].instListName := 'instances.valve';
registry.types[id - 1]._max := GC.VALVE_MAX_IDX + 1;

id := id + 1;
registry.types[id - 1].name := 'ValveReg';
registry.types[id - 1].instListName := 'instances.valveReg';
registry.types[id - 1]._max := GC.VALVE_REG_MAX_IDX + 1;

id := id + 1;
registry.types[id - 1].name := 'Drive';
registry.types[id - 1].instListName := 'instances.drive';
registry.types[id - 1]._max := GC.DRIVE_MAX_IDX + 1;

id := id + 1;
registry.types[id - 1].name := 'DriveReg';
registry.types[id - 1].instListName := 'instances.driveReg';
registry.types[id - 1]._max := GC.DRIVE_REG_MAX_IDX + 1;

id := id + 1;
registry.types[id - 1].name := 'SensorDig';
registry.types[id - 1].instListName := 'instances.sensorDig';
registry.types[id - 1]._max := GC.SENSOR_DIG_MAX_IDX + 1;

id := id + 1;
registry.types[id - 1].name := 'SensorAn';
registry.types[id - 1].instListName := 'instances.sensorAn';
registry.types[id - 1]._max := GC.SENSOR_AN_MAX_IDX + 1;

id := id + 1;

id := id + 1;
registry.types[id - 1].name := 'Hysteresis';
registry.types[id - 1].instListName := 'instances.hysteresis';
registry.types[id - 1]._max := GC.HYSTERESIS_MAX_IDX + 1;

id := id + 1; //208
registry.types[id - 1].name := 'GasFlowReg';
registry.types[id - 1].instListName := 'instances.gasFlowReg';
registry.types[id - 1]._max := GC.GAS_FLOW_REG_MAX_IDX + 1;

id := id + 1; //209
registry.types[id - 1].name := 'Cascade';
registry.types[id - 1].instListName := 'instances.cascade';
registry.types[id - 1]._max := GC.REF_MAX_IDX + 1;

id := id + 1; //210
registry.types[id - 1].name := 'Dose';
registry.types[id - 1].instListName := 'instances.dose';
registry.types[id - 1]._max := GC.DOSE_MAX_IDX + 1;

id := id + 1; //211
registry.types[id - 1].name := 'Profile';
registry.types[id - 1].instListName := 'instances.profile';
registry.types[id - 1]._max := GC.PROFILE_MAX_IDX + 1;

id := id + 1; //212
registry.types[id - 1].name := 'Ramp';
registry.types[id - 1].instListName := 'instances.ramp';
registry.types[id - 1]._max := GC.RAMP_MAX_IDX + 1;	

id := id + 1; //213
registry.types[id - 1].name := 'Route';
registry.types[id - 1].instListName := 'instances.route';
registry.types[id - 1]._max := GC.ROUTE_MAX_IDX + 1;	

id := id + 1; //214
registry.types[id - 1].name := 'Flip';
registry.types[id - 1].instListName := 'instances.flip';
registry.types[id - 1]._max := GC.FLIP_MAX_IDX + 1;

id := id + 1; //215

id := id + 1; //216

id := id + 1; //217

id := id + 1; //218

id := id + 1; //219
registry.types[id - 1].name := 'Area';
registry.types[id - 1].instListName :=  'area';
registry.types[id - 1]._max := GC.AREA_MAX_IDX + 1;

id := id + 1; //220
registry.types[id - 1].name := 'HysteresisEx';
registry.types[id - 1].instListName := 'instances.hysteresisEx';
registry.types[id - 1]._max := GC.HYSTERESISEX_MAX_IDX + 1;
END_METHOD

END_PROGRAM
